              Waypoint Home3: TCP in base x=-850.182 y=0 z=211.32 mm, rx=-2.0297 ry=2.3968 rz=0.0066 rad; joints [-14.374, -75.698, 98.757, -22.649, -284.037, -0.192] deg; TCP offset x=0.411 y=-218.298 z=37.994 mm, rx=1.558 ry=-0.1255 rz=0.1212 rad
              Waypoint Linea4_A: TCP in base x=-486.109 y=25.046 z=110.758 mm, rx=-2.0297 ry=2.3968 rz=0.0065 rad; joints [-35.513, -108.192, 141.382, -32.663, -305.184, -0.389] deg; TCP offset x=0.411 y=-218.298 z=37.994 mm, rx=1.558 ry=-0.1255 rz=0.1212 rad
              Waypoint Linea4_B: TCP in base x=-689.318 y=25.343 z=110.27 mm, rx=-2.0298 ry=2.3969 rz=0.0066 rad; joints [-21.509, -85.16, 121.882, -36.295, -291.196, -0.227] deg
              Waypoint Linea4_C: TCP in base x=-714.721 y=25.086 z=110.565 mm, rx=-2.0298 ry=2.3969 rz=0.0065 rad; joints [-20.482, -82.844, 119.204, -35.936, -290.168, -0.217] deg
              Waypoint Linea4_D: TCP in base x=-918.063 y=25.353 z=110.171 mm, rx=-2.0298 ry=2.3969 rz=0.0065 rad; joints [-14.96, -65.479, 95.824, -29.942, -284.639, -0.166] deg
              Waypoint Linea4_E: TCP in base x=-942.591 y=25.362 z=110.65 mm, rx=-2.0298 ry=2.3969 rz=0.0065 rad; joints [-14.49, -63.451, 92.661, -28.807, -284.167, -0.163] deg
              Waypoint Linea4_F: TCP in base x=-1145.81 y=25.561 z=110.408 mm, rx=-2.0298 ry=2.3969 rz=0.0066 rad; joints [-11.507, -45.055, 61.81, -16.363, -281.155, -0.146] deg
          Folder AB
            'desbaste_inicial'
            bajada_broca := p[0,0,-0.012,0,0,0]
            barrenos_menos1 := 8
            barreno_actual := 0
            Loop While (checkContinuously=false) expression=barreno_actual≤barrenos_menos1
              Folder Perforacion
                MoveL speed 100 mm/s, acceleration 500 mm/s^2 (useActiveTCP=true) feature=Base
                  internos := interpolate_pose(Linea4_A, Linea4_B, barreno_actual/barrenos_menos1)
                  Waypoint Waypoint (Variable): variable=internos
                  'desbaste_inicial'
                  bajada_broca := p[0,0,-0.012,0,0,0]
                  bajada := p[0,0,0.012,0,0,0]
                  MoveDirectionNode (selectedDirection=ZMinus toolParams=0.03, 0.035)
                    Until DISTANCE (allowActions=false deceleration=3 distanceNodeType=STOP) Distance=0.08; motionParameters(blendRadius=0)
                  Popup Message (haltProgram=false message=punto contacto alanzdo inputType=Text)
                  MoveDirectionNode (selectedDirection=ZPlus toolParams=0.003, 0.005)
                    Until DISTANCE (allowActions=false deceleration=3 distanceNodeType=STOP) Distance=0.002; motionParameters(blendRadius=0)
                  Wait Sleep waitTime=0.3
                  Set DigitalOutput pin=config_out[1]; digitalValue=1
                  Wait Sleep waitTime=0.3
                  Loop Counting (count=2) loopVariable(name=Loop_72)
                    bajar := pose_add(get_actual_tcp_pose(), bajada_broca)
                    Waypoint Waypoint (Variable): motionParameters(jointSpeed=1.047198 jointAcceleration=1.396263 cartesianSpeed=0.001 cartesianAcceleration=0.005); variable=bajar
                    subir := pose_sub(get_actual_tcp_pose(), bajada_broca)
                    Waypoint Waypoint (Variable): motionParameters(jointSpeed=1.047198 jointAcceleration=1.396263 cartesianSpeed=0.01 cartesianAcceleration=0.01); variable=subir
                    bajada_broca := pose_sub(bajada_broca, bajada)
                  MoveDirectionNode (selectedDirection=ZPlus toolParams=0.03, 0.035)
                    Until DISTANCE (allowActions=false deceleration=3 distanceNodeType=STOP) Distance=0.06; motionParameters(blendRadius=0)
                  Set DigitalOutput pin=config_out[1]; digitalValue=0
                  barreno_actual := barreno_actual+1
                  Call Quitar_broca
                  Call Poner_broca
          Folder CD
            'desbaste_inicial'
            bajada_broca := p[0,0,-0.012,0,0,0]
            barrenos_menos1 := 8
            barreno_actual := 0
            Loop While (checkContinuously=false) expression=barreno_actual≤barrenos_menos1
              Folder Perforacion
                MoveL speed 100 mm/s, acceleration 500 mm/s^2 (useActiveTCP=true) feature=Base
                  internos := interpolate_pose(Linea4_C, Linea4_D, barreno_actual/barrenos_menos1)
                  Waypoint Waypoint (Variable): variable=internos
                  'desbaste_inicial'
                  bajada_broca := p[0,0,-0.012,0,0,0]
                  bajada := p[0,0,0.012,0,0,0]
                  MoveDirectionNode (selectedDirection=ZMinus toolParams=0.03, 0.035)
                    Until DISTANCE (allowActions=false deceleration=3 distanceNodeType=STOP) Distance=0.08; motionParameters(blendRadius=0)
                  Popup Message (haltProgram=false message=punto contacto alanzdo inputType=Text)
                  MoveDirectionNode (selectedDirection=ZPlus toolParams=0.003, 0.005)
                    Until DISTANCE (allowActions=false deceleration=3 distanceNodeType=STOP) Distance=0.002; motionParameters(blendRadius=0)
                  Wait Sleep waitTime=0.3
                  Set DigitalOutput pin=config_out[1]; digitalValue=1
                  Wait Sleep waitTime=0.3
                  Loop Counting (count=2) loopVariable(name=Loop_77)
                    bajar := pose_add(get_actual_tcp_pose(), bajada_broca)
                    Waypoint Waypoint (Variable): motionParameters(jointSpeed=1.047198 jointAcceleration=1.396263 cartesianSpeed=0.001 cartesianAcceleration=0.005); variable=bajar
                    subir := pose_sub(get_actual_tcp_pose(), bajada_broca)
                    Waypoint Waypoint (Variable): motionParameters(jointSpeed=1.047198 jointAcceleration=1.396263 cartesianSpeed=0.01 cartesianAcceleration=0.01); variable=subir
                    bajada_broca := pose_sub(bajada_broca, bajada)
                  MoveDirectionNode (selectedDirection=ZPlus toolParams=0.03, 0.035)
                    Until DISTANCE (allowActions=false deceleration=3 distanceNodeType=STOP) Distance=0.06; motionParameters(blendRadius=0)
                  Set DigitalOutput pin=config_out[1]; digitalValue=0
                  barreno_actual := barreno_actual+1
                  Call Quitar_broca
                  Call Poner_broca
          Folder EF
            'desbaste_inicial'
            bajada_broca := p[0,0,-0.012,0,0,0]
            barrenos_menos1 := 8
            barreno_actual := 0
            Loop While (checkContinuously=false) expression=barreno_actual≤barrenos_menos1
              Folder Perforacion
                MoveL speed 100 mm/s, acceleration 500 mm/s^2 (useActiveTCP=true) feature=Base
                  internos := interpolate_pose(Linea4_E, Linea4_F, barreno_actual/barrenos_menos1)
                  Waypoint Waypoint (Variable): variable=internos
                  'desbaste_inicial'
                  bajada_broca := p[0,0,-0.012,0,0,0]
                  bajada := p[0,0,0.012,0,0,0]
                  MoveDirectionNode (selectedDirection=ZMinus toolParams=0.03, 0.035)
                    Until DISTANCE (allowActions=false deceleration=3 distanceNodeType=STOP) Distance=0.08; motionParameters(blendRadius=0)
                  Popup Message (haltProgram=false message=punto contacto alanzdo inputType=Text)
                  MoveDirectionNode (selectedDirection=ZPlus toolParams=0.003, 0.005)
                    Until DISTANCE (allowActions=false deceleration=3 distanceNodeType=STOP) Distance=0.002; motionParameters(blendRadius=0)
                  Wait Sleep waitTime=0.3
                  Set DigitalOutput pin=config_out[1]; digitalValue=1
                  Wait Sleep waitTime=0.3
                  Loop Counting (count=2) loopVariable(name=Loop_81)
                    bajar := pose_add(get_actual_tcp_pose(), bajada_broca)
                    Waypoint Waypoint (Variable): motionParameters(jointSpeed=1.047198 jointAcceleration=1.396263 cartesianSpeed=0.001 cartesianAcceleration=0.005); variable=bajar
                    subir := pose_sub(get_actual_tcp_pose(), bajada_broca)
                    Waypoint Waypoint (Variable): motionParameters(jointSpeed=1.047198 jointAcceleration=1.396263 cartesianSpeed=0.01 cartesianAcceleration=0.01); variable=subir
                    bajada_broca := pose_sub(bajada_broca, bajada)
                  MoveDirectionNode (selectedDirection=ZPlus toolParams=0.03, 0.035)
                    Until DISTANCE (allowActions=false deceleration=3 distanceNodeType=STOP) Distance=0.06; motionParameters(blendRadius=0)
                  Set DigitalOutput pin=config_out[1]; digitalValue=0
                  barreno_actual := barreno_actual+1
                  If barreno_actual>barrenos_menos1
                    cambiar_broca := True
                  Call Quitar_broca
                  Call Poner_broca
        Popup Message (haltProgram=false message=Linea4 con media Terminada! inputType=Text)
      Folder Broca_3
        Folder Linea3
          Folder Marcar_puntos
            MoveL speed 100 mm/s, acceleration 500 mm/s^2 (useActiveTCP=true) feature=Base
              Waypoint Home3: TCP in base x=-850.182 y=0 z=211.32 mm, rx=-2.0297 ry=2.3968 rz=0.0066 rad; joints [-14.374, -75.698, 98.757, -22.649, -284.037, -0.192] deg; TCP offset x=0.411 y=-218.298 z=37.994 mm, rx=1.558 ry=-0.1255 rz=0.1212 rad
              Folder var
                barrenos_hechos := 0
                eje7 := 3
                cambiar_broca := False
                iniciando_prog := True
              Call Poner_broca
              Waypoint Linea3_A: TCP in base x=-486.114 y=-381.655 z=110.21 mm, rx=-2.0297 ry=2.3968 rz=0.0065 rad; joints [28.783, -88.014, 124.97, -36.558, -240.905, 0.122] deg; TCP offset x=0.411 y=-218.298 z=37.994 mm, rx=1.558 ry=-0.1255 rz=0.1212 rad
              Waypoint Linea3_B: TCP in base x=-689.31 y=-380.791 z=110.221 mm, rx=-2.0297 ry=2.3969 rz=0.0065 rad; joints [20.056, -74.462, 108.7, -33.857, -249.629, 0.064] deg
              Waypoint Linea3_C: TCP in base x=-714.73 y=-381.227 z=110.547 mm, rx=-2.0298 ry=2.3969 rz=0.0065 rad; joints [19.334, -72.698, 106.253, -33.176, -250.351, 0.061] deg
              Waypoint Linea3_D: TCP in base x=-917.837 y=-380.542 z=110.222 mm, rx=-2.0298 ry=2.3969 rz=0.0065 rad; joints [14.731, -57.949, 83.951, -25.628, -254.939, 0.03] deg
              Waypoint Linea3_E: TCP in base x=-943.23 y=-380.75 z=110.26 mm, rx=-2.0297 ry=2.3969 rz=0.0065 rad; joints [14.315, -55.955, 80.664, -24.335, -255.35, 0.027] deg
              Waypoint Linea3_F: TCP in base x=-1146.085 y=-380.44 z=110.221 mm, rx=-2.0297 ry=2.397 rz=0.0066 rad; joints [11.572, -37.03, 47.136, -9.737, -258.055, 0.004] deg
          Folder AB
            'desbaste_inicial'
            bajada_broca := p[0,0,-0.024,0,0,0]
            barrenos_menos1 := 8
            barreno_actual := 5
            Loop While (checkContinuously=false) expression=barreno_actual≤barrenos_menos1
              Folder Perforacion
                MoveL speed 100 mm/s, acceleration 500 mm/s^2 (useActiveTCP=true) feature=Base
                  internos := interpolate_pose(Linea3_A, Linea3_B, barreno_actual/barrenos_menos1)
                  Waypoint Waypoint (Variable): variable=internos
                  'desbaste_inicial'
                  bajada_broca := p[0,0,-0.024,0,0,0]
                  bajada := p[0,0,0.024,0,0,0]
                  MoveDirectionNode (selectedDirection=ZMinus toolParams=0.03, 0.035)
                    Until DISTANCE (allowActions=false deceleration=3 distanceNodeType=STOP) Distance=0.083; motionParameters(blendRadius=0)
                  Popup Message (haltProgram=false message=punto contacto alanzdo inputType=Text)
                  MoveDirectionNode (selectedDirection=ZPlus toolParams=0.003, 0.005)
                    Until DISTANCE (allowActions=false deceleration=3 distanceNodeType=STOP) Distance=0.002; motionParameters(blendRadius=0)
                  Wait Sleep waitTime=0.3
                  Set DigitalOutput pin=config_out[1]; digitalValue=1
                  Wait Sleep waitTime=0.3
                  Loop Counting (count=1) loopVariable=Loop_86
                    bajar := pose_add(get_actual_tcp_pose(), bajada_broca)
                    Waypoint Waypoint (Variable): motionParameters(jointSpeed=1.047198 jointAcceleration=1.396263 cartesianSpeed=0.001 cartesianAcceleration=0.005); variable=bajar
                    subir := pose_sub(get_actual_tcp_pose(), bajada_broca)
                    Waypoint Waypoint (Variable): motionParameters(jointSpeed=1.047198 jointAcceleration=1.396263 cartesianSpeed=0.01 cartesianAcceleration=0.01); variable=subir
                    bajada_broca := pose_sub(bajada_broca, bajada)
                  MoveDirectionNode (selectedDirection=ZPlus toolParams=0.03, 0.035)
                    Until DISTANCE (allowActions=false deceleration=3 distanceNodeType=STOP) Distance=0.06; motionParameters(blendRadius=0)
                  Set DigitalOutput pin=config_out[1]; digitalValue=0
                  barreno_actual := barreno_actual+1
                  Call Quitar_broca
                  Call Poner_broca
          Folder CD
            'desbaste_inicial'
            bajada_broca := p[0,0,-0.024,0,0,0]
            barrenos_menos1 := 8
            barreno_actual := 0
            Loop While (checkContinuously=false) expression=barreno_actual≤barrenos_menos1
              Folder Perforacion
                MoveL speed 100 mm/s, acceleration 500 mm/s^2 (useActiveTCP=true) feature=Base
                  internos := interpolate_pose(Linea3_C, Linea3_D, barreno_actual/barrenos_menos1)
                  Waypoint Waypoint (Variable): variable=internos
                  'desbaste_inicial'
                  bajada_broca := p[0,0,-0.024,0,0,0]
                  bajada := p[0,0,0.024,0,0,0]
                  MoveDirectionNode (selectedDirection=ZMinus toolParams=0.03, 0.035)
                    Until DISTANCE (allowActions=false deceleration=3 distanceNodeType=STOP) Distance=0.083; motionParameters(blendRadius=0)
                  Popup Message (haltProgram=false message=punto contacto alanzdo inputType=Text)
                  MoveDirectionNode (selectedDirection=ZPlus toolParams=0.003, 0.005)
                    Until DISTANCE (allowActions=false deceleration=3 distanceNodeType=STOP) Distance=0.002; motionParameters(blendRadius=0)
                  Wait Sleep waitTime=0.3
                  Set DigitalOutput pin=config_out[1]; digitalValue=1
                  Wait Sleep waitTime=0.3
                  Loop Counting (count=1) loopVariable(name=Loop_91)
                    bajar := pose_add(get_actual_tcp_pose(), bajada_broca)
                    Waypoint Waypoint (Variable): motionParameters(jointSpeed=1.047198 jointAcceleration=1.396263 cartesianSpeed=0.001 cartesianAcceleration=0.005); variable=bajar
                    subir := pose_sub(get_actual_tcp_pose(), bajada_broca)
                    Waypoint Waypoint (Variable): motionParameters(jointSpeed=1.047198 jointAcceleration=1.396263 cartesianSpeed=0.01 cartesianAcceleration=0.01); variable=subir
                    bajada_broca := pose_sub(bajada_broca, bajada)
                  MoveDirectionNode (selectedDirection=ZPlus toolParams=0.03, 0.035)
                    Until DISTANCE (allowActions=false deceleration=3 distanceNodeType=STOP) Distance=0.06; motionParameters(blendRadius=0)
                  Set DigitalOutput pin=config_out[1]; digitalValue=0
                  barreno_actual := barreno_actual+1
                  Call Quitar_broca
                  Call Poner_broca
          Folder EF
            'desbaste_inicial'
            bajada_broca := p[0,0,-0.024,0,0,0]
            barrenos_menos1 := 8
            barreno_actual := 0
            Loop While (checkContinuously=false) expression=barreno_actual≤barrenos_menos1
              Folder Perforacion
                MoveL speed 100 mm/s, acceleration 500 mm/s^2 (useActiveTCP=true) feature=Base
                  internos := interpolate_pose(Linea3_E, Linea3_F, barreno_actual/barrenos_menos1)
                  Waypoint Waypoint (Variable): variable=internos
                  'desbaste_inicial'
                  bajada_broca := p[0,0,-0.024,0,0,0]
                  bajada := p[0,0,0.024,0,0,0]
                  MoveDirectionNode (selectedDirection=ZMinus toolParams=0.03, 0.035)
                    Until DISTANCE (allowActions=false deceleration=3 distanceNodeType=STOP) Distance=0.083; motionParameters(blendRadius=0)
                  Popup Message (haltProgram=false message=punto contacto alanzdo inputType=Text)
                  MoveDirectionNode (selectedDirection=ZPlus toolParams=0.003, 0.005)
                    Until DISTANCE (allowActions=false deceleration=3 distanceNodeType=STOP) Distance=0.002; motionParameters(blendRadius=0)
                  Wait Sleep waitTime=0.3
                  Set DigitalOutput pin=config_out[1]; digitalValue=1
                  Wait Sleep waitTime=0.3
                  Loop Counting (count=1) loopVariable=Loop_100
                    bajar := pose_add(get_actual_tcp_pose(), bajada_broca)
                    Waypoint Waypoint (Variable): motionParameters(jointSpeed=1.047198 jointAcceleration=1.396263 cartesianSpeed=0.001 cartesianAcceleration=0.005); variable=bajar
                    subir := pose_sub(get_actual_tcp_pose(), bajada_broca)
                    Waypoint Waypoint (Variable): motionParameters(jointSpeed=1.047198 jointAcceleration=1.396263 cartesianSpeed=0.01 cartesianAcceleration=0.01); variable=subir
                    bajada_broca := pose_sub(bajada_broca, bajada)
                  MoveDirectionNode (selectedDirection=ZPlus toolParams=0.03, 0.035)
                    Until DISTANCE (allowActions=false deceleration=3 distanceNodeType=STOP) Distance=0.06; motionParameters(blendRadius=0)
                  Set DigitalOutput pin=config_out[1]; digitalValue=0
                  barreno_actual := barreno_actual+1
                  Call Quitar_broca
                  Call Poner_broca
        Popup Message (haltProgram=false message=Linea3 con full Terminada! inputType=Text)
        Folder Linea4
          Folder Marcar_puntos
            MoveL speed 100 mm/s, acceleration 500 mm/s^2 (useActiveTCP=true) feature=Base
              Waypoint Home3: TCP in base x=-850.182 y=0 z=211.32 mm, rx=-2.0297 ry=2.3968 rz=0.0066 rad; joints [-14.374, -75.698, 98.757, -22.649, -284.037, -0.192] deg; TCP offset x=0.411 y=-218.298 z=37.994 mm, rx=1.558 ry=-0.1255 rz=0.1212 rad
              Waypoint Linea4_A: TCP in base x=-486.109 y=25.046 z=110.758 mm, rx=-2.0297 ry=2.3968 rz=0.0065 rad; joints [-35.513, -108.192, 141.382, -32.663, -305.184, -0.389] deg; TCP offset x=0.411 y=-218.298 z=37.994 mm, rx=1.558 ry=-0.1255 rz=0.1212 rad
              Waypoint Linea4_B: TCP in base x=-689.318 y=25.343 z=110.27 mm, rx=-2.0298 ry=2.3969 rz=0.0066 rad; joints [-21.509, -85.16, 121.882, -36.295, -291.196, -0.227] deg
              Waypoint Linea4_C: TCP in base x=-714.721 y=25.086 z=110.565 mm, rx=-2.0298 ry=2.3969 rz=0.0065 rad; joints [-20.482, -82.844, 119.204, -35.936, -290.168, -0.217] deg
              Waypoint Linea4_D: TCP in base x=-918.063 y=25.353 z=110.171 mm, rx=-2.0298 ry=2.3969 rz=0.0065 rad; joints [-14.96, -65.479, 95.824, -29.942, -284.639, -0.166] deg
              Waypoint Linea4_E: TCP in base x=-942.591 y=25.362 z=110.65 mm, rx=-2.0298 ry=2.3969 rz=0.0065 rad; joints [-14.49, -63.451, 92.661, -28.807, -284.167, -0.163] deg
              Waypoint Linea4_F: TCP in base x=-1145.81 y=25.561 z=110.408 mm, rx=-2.0298 ry=2.3969 rz=0.0066 rad; joints [-11.507, -45.055, 61.81, -16.363, -281.155, -0.146] deg
          Folder AB
            'desbaste_inicial'
            bajada_broca := p[0,0,-0.024,0,0,0]
            barrenos_menos1 := 8
            barreno_actual := 0
            Loop While (checkContinuously=false) expression=barreno_actual≤barrenos_menos1
              Folder Perforacion
                MoveL speed 100 mm/s, acceleration 500 mm/s^2 (useActiveTCP=true) feature=Base
                  internos := interpolate_pose(Linea4_A, Linea4_B, barreno_actual/barrenos_menos1)
                  Waypoint Waypoint (Variable): variable=internos
                  'desbaste_inicial'
                  bajada_broca := p[0,0,-0.024,0,0,0]
                  bajada := p[0,0,0.024,0,0,0]
                  MoveDirectionNode (selectedDirection=ZMinus toolParams=0.03, 0.035)
                    Until DISTANCE (allowActions=false deceleration=3 distanceNodeType=STOP) Distance=0.083; motionParameters(blendRadius=0)
                  Popup Message (haltProgram=false message=punto contacto alanzdo inputType=Text)
                  MoveDirectionNode (selectedDirection=ZPlus toolParams=0.003, 0.005)
                    Until DISTANCE (allowActions=false deceleration=3 distanceNodeType=STOP) Distance=0.002; motionParameters(blendRadius=0)
                  Wait Sleep waitTime=0.3
                  Set DigitalOutput pin=config_out[1]; digitalValue=1
                  Wait Sleep waitTime=0.3
                  Loop Counting (count=1) loopVariable(name=Loop_120)
                    bajar := pose_add(get_actual_tcp_pose(), bajada_broca)
                    Waypoint Waypoint (Variable): motionParameters(jointSpeed=1.047198 jointAcceleration=1.396263 cartesianSpeed=0.001 cartesianAcceleration=0.005); variable=bajar
                    subir := pose_sub(get_actual_tcp_pose(), bajada_broca)
                    Waypoint Waypoint (Variable): motionParameters(jointSpeed=1.047198 jointAcceleration=1.396263 cartesianSpeed=0.01 cartesianAcceleration=0.01); variable=subir
                    bajada_broca := pose_sub(bajada_broca, bajada)
                  MoveDirectionNode (selectedDirection=ZPlus toolParams=0.03, 0.035)
                    Until DISTANCE (allowActions=false deceleration=3 distanceNodeType=STOP) Distance=0.06; motionParameters(blendRadius=0)
                  Set DigitalOutput pin=config_out[1]; digitalValue=0
                  barreno_actual := barreno_actual+1
                  Call Quitar_broca
                  Call Poner_broca
          Folder CD
            'desbaste_inicial'
            bajada_broca := p[0,0,-0.024,0,0,0]
            barrenos_menos1 := 8
            barreno_actual := 0
            Loop While (checkContinuously=false) expression=barreno_actual≤barrenos_menos1
              Folder Perforacion
                MoveL speed 100 mm/s, acceleration 500 mm/s^2 (useActiveTCP=true) feature=Base
                  internos := interpolate_pose(Linea4_C, Linea4_D, barreno_actual/barrenos_menos1)
                  Waypoint Waypoint (Variable): variable=internos
                  'desbaste_inicial'
                  bajada_broca := p[0,0,-0.024,0,0,0]
                  bajada := p[0,0,0.024,0,0,0]
                  MoveDirectionNode (selectedDirection=ZMinus toolParams=0.03, 0.035)
                    Until DISTANCE (allowActions=false deceleration=3 distanceNodeType=STOP) Distance=0.083; motionParameters(blendRadius=0)
                  Popup Message (haltProgram=false message=punto contacto alanzdo inputType=Text)
                  MoveDirectionNode (selectedDirection=ZPlus toolParams=0.003, 0.005)
                    Until DISTANCE (allowActions=false deceleration=3 distanceNodeType=STOP) Distance=0.002; motionParameters(blendRadius=0)
                  Wait Sleep waitTime=0.3
                  Set DigitalOutput pin=config_out[1]; digitalValue=1
                  Wait Sleep waitTime=0.3
                  Loop Counting (count=1) loopVariable=Loop_123
                    bajar := pose_add(get_actual_tcp_pose(), bajada_broca)
                    Waypoint Waypoint (Variable): motionParameters(jointSpeed=1.047198 jointAcceleration=1.396263 cartesianSpeed=0.001 cartesianAcceleration=0.005); variable=bajar
                    subir := pose_sub(get_actual_tcp_pose(), bajada_broca)
                    Waypoint Waypoint (Variable): motionParameters(jointSpeed=1.047198 jointAcceleration=1.396263 cartesianSpeed=0.01 cartesianAcceleration=0.01); variable=subir
                    bajada_broca := pose_sub(bajada_broca, bajada)
                  MoveDirectionNode (selectedDirection=ZPlus toolParams=0.03, 0.035)
                    Until DISTANCE (allowActions=false deceleration=3 distanceNodeType=STOP) Distance=0.06; motionParameters(blendRadius=0)
                  Set DigitalOutput pin=config_out[1]; digitalValue=0
                  barreno_actual := barreno_actual+1
                  Call Quitar_broca
                  Call Poner_broca
          Folder EF
            'desbaste_inicial'
            bajada_broca := p[0,0,-0.024,0,0,0]
            barrenos_menos1 := 8
            barreno_actual := 0
            Loop While (checkContinuously=false) expression=barreno_actual≤barrenos_menos1
              Folder Perforacion
                MoveL speed 100 mm/s, acceleration 500 mm/s^2 (useActiveTCP=true) feature=Base
                  internos := interpolate_pose(Linea4_E, Linea4_F, barreno_actual/barrenos_menos1)
                  Waypoint Waypoint (Variable): variable=internos
                  'desbaste_inicial'
                  bajada_broca := p[0,0,-0.024,0,0,0]
                  bajada := p[0,0,0.024,0,0,0]
                  MoveDirectionNode (selectedDirection=ZMinus toolParams=0.03, 0.035)
                    Until DISTANCE (allowActions=false deceleration=3 distanceNodeType=STOP) Distance=0.083; motionParameters(blendRadius=0)
                  Popup Message (haltProgram=false message=punto contacto alanzdo inputType=Text)
                  MoveDirectionNode (selectedDirection=ZPlus toolParams=0.003, 0.005)
                    Until DISTANCE (allowActions=false deceleration=3 distanceNodeType=STOP) Distance=0.002; motionParameters(blendRadius=0)
                  Wait Sleep waitTime=0.3
                  Set DigitalOutput pin=config_out[1]; digitalValue=1
                  Wait Sleep waitTime=0.3
                  Loop Counting (count=1) loopVariable=Loop_125
                    bajar := pose_add(get_actual_tcp_pose(), bajada_broca)
                    Waypoint Waypoint (Variable): motionParameters(jointSpeed=1.047198 jointAcceleration=1.396263 cartesianSpeed=0.001 cartesianAcceleration=0.005); variable=bajar
                    subir := pose_sub(get_actual_tcp_pose(), bajada_broca)
                    Waypoint Waypoint (Variable): motionParameters(jointSpeed=1.047198 jointAcceleration=1.396263 cartesianSpeed=0.01 cartesianAcceleration=0.01); variable=subir
                    bajada_broca := pose_sub(bajada_broca, bajada)
                  MoveDirectionNode (selectedDirection=ZPlus toolParams=0.03, 0.035)
                    Until DISTANCE (allowActions=false deceleration=3 distanceNodeType=STOP) Distance=0.06; motionParameters(blendRadius=0)
                  Set DigitalOutput pin=config_out[1]; digitalValue=0
                  barreno_actual := barreno_actual+1
                  If barreno_actual>barrenos_menos1
                    cambiar_broca := True
                  Call Quitar_broca
                  Call Poner_broca
        Popup Message (haltProgram=false message=Linea4 con full Terminada! inputType=Text)
    SuppressedNode
      Folder 720
        Folder Broca_1
          Folder Linea5
            Folder Marcar_puntos
              MoveL speed 100 mm/s, acceleration 500 mm/s^2 (useActiveTCP=true) feature=Base
                Waypoint Home3: TCP in base x=-850.182 y=0 z=211.32 mm, rx=-2.0297 ry=2.3968 rz=0.0066 rad; joints [-14.374, -75.698, 98.757, -22.649, -284.037, -0.192] deg; TCP offset x=0.411 y=-218.298 z=37.994 mm, rx=1.558 ry=-0.1255 rz=0.1212 rad
                Waypoint Linea5_A: TCP in base x=-663.778 y=-510.056 z=80.075 mm, rx=3.1116 ry=-0.3921 rz=0.0087 rad; joints [15.224, -65.782, 99.916, -33.468, -339.581, -0.139] deg; TCP offset x=0.411 y=-218.298 z=37.994 mm, rx=1.558 ry=-0.1255 rz=0.1212 rad
                Waypoint Linea5_B: TCP in base x=-1154.197 y=-507.911 z=80.256 mm, rx=-2.6466 ry=1.68 rz=0.0007 rad; joints [13.333, -29.304, 35.323, -5.09, -290.95, -0.372] deg
            Folder AB
              'desbaste_inicial'
              bajada_broca := p[0,0,-0.008,0,0,0]
              barrenos_menos1 := 19
              barreno_actual := 0
              Loop While (checkContinuously=false) expression=barreno_actual≤barrenos_menos1
                Folder Perforacion
                  MoveL speed 100 mm/s, acceleration 500 mm/s^2 (useActiveTCP=true) feature=Base
                    internos := interpolate_pose(Linea5_A, Linea5_B, barreno_actual/barrenos_menos1)
                    Waypoint Waypoint (Variable): variable=internos
                    'desbaste_inicial'
                    bajada_broca := p[0,0,-0.008,0,0,0]
                    bajada := p[0,0,0.008,0,0,0]
                    MoveDirectionNode (selectedDirection=ZMinus toolParams=0.007, 0.005)
                      Until TOOL_CONTACT_DETECTION (allowActions=false retraction=0 decelerationAcceleration=0.001 decelerationAngularAcceleration=34.906585)
                    Popup Message (haltProgram=false message=punto contacto alanzdo inputType=Text)
                    SuppressedNode
                      MoveDirectionNode (selectedDirection=ZPlus toolParams=0.003, 0.005)
                        Until DISTANCE (allowActions=false deceleration=3 distanceNodeType=STOP) Distance=0.002; motionParameters(blendRadius=0)
                    SuppressedNode
                      Wait Sleep waitTime=0.3
                    SuppressedNode
                      Set DigitalOutput pin=config_out[1]; digitalValue=1
                    SuppressedNode
                      Wait Sleep waitTime=0.3
                    SuppressedNode
                      Loop Counting (count=3) loopVariable(name=Loop_55)
                        bajar := pose_add(get_actual_tcp_pose(), bajada_broca)
                        Waypoint Waypoint (Variable): motionParameters(jointSpeed=1.047198 jointAcceleration=1.396263 cartesianSpeed=0.001 cartesianAcceleration=0.005); variable=bajar
                        subir := pose_sub(get_actual_tcp_pose(), bajada_broca)
                        Waypoint Waypoint (Variable): motionParameters(jointSpeed=1.047198 jointAcceleration=1.396263 cartesianSpeed=0.01 cartesianAcceleration=0.01); variable=subir
                        bajada_broca := pose_sub(bajada_broca, bajada)
                    MoveDirectionNode (selectedDirection=ZPlus toolParams=0.03, 0.035)
                      Until DISTANCE (allowActions=false deceleration=3 distanceNodeType=STOP) Distance=0.15; motionParameters(blendRadius=0)
                    Set DigitalOutput pin=config_out[1]; digitalValue=0
                    barreno_actual := barreno_actual+1
                    SuppressedNode
                      Call Quitar_broca
                    SuppressedNode
                      Call Poner_broca
            SuppressedNode
              Folder CD
                'desbaste_inicial'
                bajada_broca := p[0,0,-0.008,0,0,0]
                barrenos_menos1 := 8
                barreno_actual := 0
                Loop While (checkContinuously=false) expression=barreno_actual≤barrenos_menos1
                  Folder Perforacion
                    MoveL speed 100 mm/s, acceleration 500 mm/s^2 (useActiveTCP=true) feature=Base
                      internos := interpolate_pose(Linea3_C, Linea3_D, barreno_actual/barrenos_menos1)
                      Waypoint Waypoint (Variable): variable=internos
                      'desbaste_inicial'
                      bajada_broca := p[0,0,-0.008,0,0,0]
                      bajada := p[0,0,0.008,0,0,0]
                      MoveDirectionNode (selectedDirection=ZMinus toolParams=0.02, 0.015)
                        Until DISTANCE (allowActions=false deceleration=3 distanceNodeType=STOP) Distance=0.055; motionParameters(blendRadius=0)
                      Popup Message (haltProgram=false message=punto contacto alanzdo inputType=Text)
                      MoveDirectionNode (selectedDirection=ZPlus toolParams=0.003, 0.005)
                        Until DISTANCE (allowActions=false deceleration=3 distanceNodeType=STOP) Distance=0.002; motionParameters(blendRadius=0)
                      Wait Sleep waitTime=0.3
                      Set DigitalOutput pin=config_out[1]; digitalValue=1
                      Wait Sleep waitTime=0.3
                      Loop Counting (count=3) loopVariable(name=Loop_57)
                        bajar := pose_add(get_actual_tcp_pose(), bajada_broca)
                        Waypoint Waypoint (Variable): motionParameters(jointSpeed=1.047198 jointAcceleration=1.396263 cartesianSpeed=0.001 cartesianAcceleration=0.005); variable=bajar
                        subir := pose_sub(get_actual_tcp_pose(), bajada_broca)
                        Waypoint Waypoint (Variable): motionParameters(jointSpeed=1.047198 jointAcceleration=1.396263 cartesianSpeed=0.01 cartesianAcceleration=0.01); variable=subir
                        bajada_broca := pose_sub(bajada_broca, bajada)
                      MoveDirectionNode (selectedDirection=ZPlus toolParams=0.03, 0.035)
                        Until DISTANCE (allowActions=false deceleration=3 distanceNodeType=STOP) Distance=0.06; motionParameters(blendRadius=0)
                      Set DigitalOutput pin=config_out[1]; digitalValue=0
                      barreno_actual := barreno_actual+1
                      SuppressedNode
                        Call Quitar_broca
                      SuppressedNode
                        Call Poner_broca
            SuppressedNode
              Folder EF
                'desbaste_inicial'
                bajada_broca := p[0,0,-0.008,0,0,0]
                barrenos_menos1 := 8
                barreno_actual := 0
                Loop While (checkContinuously=false) expression=barreno_actual≤barrenos_menos1
                  Folder Perforacion
                    MoveL speed 100 mm/s, acceleration 500 mm/s^2 (useActiveTCP=true) feature=Base
                      internos := interpolate_pose(Linea3_E, Linea3_F, barreno_actual/barrenos_menos1)
                      Waypoint Waypoint (Variable): variable=internos
                      'desbaste_inicial'
                      bajada_broca := p[0,0,-0.008,0,0,0]
                      bajada := p[0,0,0.008,0,0,0]
                      MoveDirectionNode (selectedDirection=ZMinus toolParams=0.02, 0.015)
                        Until DISTANCE (allowActions=false deceleration=3 distanceNodeType=STOP) Distance=0.055; motionParameters(blendRadius=0)
                      Popup Message (haltProgram=false message=punto contacto alanzdo inputType=Text)
                      MoveDirectionNode (selectedDirection=ZPlus toolParams=0.003, 0.005)
                        Until DISTANCE (allowActions=false deceleration=3 distanceNodeType=STOP) Distance=0.002; motionParameters(blendRadius=0)
                      Wait Sleep waitTime=0.3
                      Set DigitalOutput pin=config_out[1]; digitalValue=1
                      Wait Sleep waitTime=0.3
                      Loop Counting (count=3) loopVariable(name=Loop_59)
                        bajar := pose_add(get_actual_tcp_pose(), bajada_broca)
                        Waypoint Waypoint (Variable): motionParameters(jointSpeed=1.047198 jointAcceleration=1.396263 cartesianSpeed=0.001 cartesianAcceleration=0.005); variable=bajar
                        subir := pose_sub(get_actual_tcp_pose(), bajada_broca)
                        Waypoint Waypoint (Variable): motionParameters(jointSpeed=1.047198 jointAcceleration=1.396263 cartesianSpeed=0.01 cartesianAcceleration=0.01); variable=subir
                        bajada_broca := pose_sub(bajada_broca, bajada)
                      MoveDirectionNode (selectedDirection=ZPlus toolParams=0.03, 0.035)
                        Until DISTANCE (allowActions=false deceleration=3 distanceNodeType=STOP) Distance=0.06; motionParameters(blendRadius=0)
                      Set DigitalOutput pin=config_out[1]; digitalValue=0
                      barreno_actual := barreno_actual+1
                      SuppressedNode
                        Call Quitar_broca
                      SuppressedNode
                        Call Poner_broca
          Popup Message (haltProgram=false message=Linea5 con chica Terminada! inputType=Text)
          Folder Linea6
            Folder Marcar_puntos
              MoveL speed 100 mm/s, acceleration 500 mm/s^2 (useActiveTCP=true) feature=Base
                Waypoint Home3: TCP in base x=-850.182 y=0 z=211.32 mm, rx=-2.0297 ry=2.3968 rz=0.0066 rad; joints [-14.374, -75.698, 98.757, -22.649, -284.037, -0.192] deg; TCP offset x=0.411 y=-218.298 z=37.994 mm, rx=1.558 ry=-0.1255 rz=0.1212 rad
                Waypoint Linea4_A: TCP in base x=-483.35 y=19.133 z=80.413 mm, rx=-2.0297 ry=2.3968 rz=0.0066 rad; joints [-34.857, -105.949, 143.743, -37.281, -304.535, -0.37] deg
                Waypoint Linea4_B: TCP in base x=-685.405 y=19.216 z=80.605 mm, rx=-2.0297 ry=2.3968 rz=0.0066 rad; joints [-21.02, -83.488, 123.782, -39.869, -290.712, -0.217] deg
                Waypoint Linea4_C: TCP in base x=-711.768 y=19.56 z=80.904 mm, rx=-2.0297 ry=2.3968 rz=0.0066 rad; joints [-20.032, -81.151, 120.968, -39.396, -289.723, -0.208] deg
                Waypoint Linea4_D: TCP in base x=-914.58 y=19.801 z=80.703 mm, rx=-2.0297 ry=2.3968 rz=0.0066 rad; joints [-14.612, -64.317, 97.516, -32.795, -284.295, -0.166] deg
                Waypoint Linea4_E: TCP in base x=-939.799 y=20.701 z=80.126 mm, rx=-2.0297 ry=2.3968 rz=0.0066 rad; joints [-14.202, -62.236, 94.311, -31.673, -283.882, -0.163] deg
                Waypoint Linea4_F: TCP in base x=-1143.008 y=20.924 z=80.361 mm, rx=-2.0297 ry=2.3968 rz=0.0066 rad; joints [-11.271, -44.369, 63.742, -18.977, -280.923, -0.147] deg
            Folder AB
              'desbaste_inicial'
              bajada_broca := p[0,0,-0.008,0,0,0]
              barrenos_menos1 := 8
              barreno_actual := 0
              Loop While (checkContinuously=false) expression=barreno_actual≤barrenos_menos1
                Folder Perforacion
                  MoveL speed 100 mm/s, acceleration 500 mm/s^2 (useActiveTCP=true) feature=Base
                    internos := interpolate_pose(Linea4_A, Linea4_B, barreno_actual/barrenos_menos1)
                    Waypoint Waypoint (Variable): variable=internos
                    'desbaste_inicial'
                    bajada_broca := p[0,0,-0.008,0,0,0]
                    bajada := p[0,0,0.008,0,0,0]
                    MoveDirectionNode (selectedDirection=ZMinus toolParams=0.02, 0.015)
                      Until DISTANCE (allowActions=false deceleration=3 distanceNodeType=STOP) Distance=0.055; motionParameters(blendRadius=0)
                    Popup Message (haltProgram=false message=punto contacto alanzdo inputType=Text)
                    MoveDirectionNode (selectedDirection=ZPlus toolParams=0.003, 0.005)
                      Until DISTANCE (allowActions=false deceleration=3 distanceNodeType=STOP) Distance=0.002; motionParameters(blendRadius=0)
                    Wait Sleep waitTime=0.3
                    Set DigitalOutput pin=config_out[1]; digitalValue=1
                    Wait Sleep waitTime=0.3
                    Loop Counting (count=3) loopVariable=Loop_61
                      bajar := pose_add(get_actual_tcp_pose(), bajada_broca)
                      Waypoint Waypoint (Variable): motionParameters(jointSpeed=1.047198 jointAcceleration=1.396263 cartesianSpeed=0.001 cartesianAcceleration=0.005); variable=bajar
                      subir := pose_sub(get_actual_tcp_pose(), bajada_broca)
                      Waypoint Waypoint (Variable): motionParameters(jointSpeed=1.047198 jointAcceleration=1.396263 cartesianSpeed=0.01 cartesianAcceleration=0.01); variable=subir
                      bajada_broca := pose_sub(bajada_broca, bajada)
                    MoveDirectionNode (selectedDirection=ZPlus toolParams=0.03, 0.035)
                      Until DISTANCE (allowActions=false deceleration=3 distanceNodeType=STOP) Distance=0.06; motionParameters(blendRadius=0)
                    Set DigitalOutput pin=config_out[1]; digitalValue=0
                    barreno_actual := barreno_actual+1
                    SuppressedNode
                      Call Quitar_broca
                    SuppressedNode
                      Call Poner_broca
            Folder CD
              'desbaste_inicial'
              bajada_broca := p[0,0,-0.008,0,0,0]
              barrenos_menos1 := 8
              barreno_actual := 0
              Loop While (checkContinuously=false) expression=barreno_actual≤barrenos_menos1
                Folder Perforacion
                  MoveL speed 100 mm/s, acceleration 500 mm/s^2 (useActiveTCP=true) feature=Base
                    internos := interpolate_pose(Linea4_C, Linea4_D, barreno_actual/barrenos_menos1)
                    Waypoint Waypoint (Variable): variable=internos
                    'desbaste_inicial'
                    bajada_broca := p[0,0,-0.008,0,0,0]
                    bajada := p[0,0,0.008,0,0,0]
                    MoveDirectionNode (selectedDirection=ZMinus toolParams=0.02, 0.015)
                      Until DISTANCE (allowActions=false deceleration=3 distanceNodeType=STOP) Distance=0.055; motionParameters(blendRadius=0)
                    Popup Message (haltProgram=false message=punto contacto alanzdo inputType=Text)
                    MoveDirectionNode (selectedDirection=ZPlus toolParams=0.003, 0.005)
                      Until DISTANCE (allowActions=false deceleration=3 distanceNodeType=STOP) Distance=0.002; motionParameters(blendRadius=0)
                    Wait Sleep waitTime=0.3
                    Set DigitalOutput pin=config_out[1]; digitalValue=1
                    Wait Sleep waitTime=0.3
                    Loop Counting (count=3) loopVariable=Loop_63
                      bajar := pose_add(get_actual_tcp_pose(), bajada_broca)
                      Waypoint Waypoint (Variable): motionParameters(jointSpeed=1.047198 jointAcceleration=1.396263 cartesianSpeed=0.001 cartesianAcceleration=0.005); variable=bajar
                      subir := pose_sub(get_actual_tcp_pose(), bajada_broca)
                      Waypoint Waypoint (Variable): motionParameters(jointSpeed=1.047198 jointAcceleration=1.396263 cartesianSpeed=0.01 cartesianAcceleration=0.01); variable=subir
                      bajada_broca := pose_sub(bajada_broca, bajada)
                    MoveDirectionNode (selectedDirection=ZPlus toolParams=0.03, 0.035)
                      Until DISTANCE (allowActions=false deceleration=3 distanceNodeType=STOP) Distance=0.06; motionParameters(blendRadius=0)
                    Set DigitalOutput pin=config_out[1]; digitalValue=0
                    barreno_actual := barreno_actual+1
                    SuppressedNode
                      Call Quitar_broca
                    SuppressedNode
                      Call Poner_broca
            Folder EF
              'desbaste_inicial'
              bajada_broca := p[0,0,-0.008,0,0,0]
              barrenos_menos1 := 8
              barreno_actual := 0
              Loop While (checkContinuously=false) expression=barreno_actual≤barrenos_menos1
                Folder Perforacion
                  MoveL speed 100 mm/s, acceleration 500 mm/s^2 (useActiveTCP=true) feature=Base
                    internos := interpolate_pose(Linea4_E, Linea4_F, barreno_actual/barrenos_menos1)
                    Waypoint Waypoint (Variable): variable=internos
                    'desbaste_inicial'
                    bajada_broca := p[0,0,-0.008,0,0,0]
                    bajada := p[0,0,0.008,0,0,0]
                    MoveDirectionNode (selectedDirection=ZMinus toolParams=0.02, 0.015)
                      Until DISTANCE (allowActions=false deceleration=3 distanceNodeType=STOP) Distance=0.055; motionParameters(blendRadius=0)
                    Popup Message (haltProgram=false message=punto contacto alanzdo inputType=Text)
                    MoveDirectionNode (selectedDirection=ZPlus toolParams=0.003, 0.005)
                      Until DISTANCE (allowActions=false deceleration=3 distanceNodeType=STOP) Distance=0.002; motionParameters(blendRadius=0)
                    Wait Sleep waitTime=0.3
                    Set DigitalOutput pin=config_out[1]; digitalValue=1
                    Wait Sleep waitTime=0.3
                    Loop Counting (count=3) loopVariable=Loop_65
                      bajar := pose_add(get_actual_tcp_pose(), bajada_broca)
                      Waypoint Waypoint (Variable): motionParameters(jointSpeed=1.047198 jointAcceleration=1.396263 cartesianSpeed=0.001 cartesianAcceleration=0.005); variable=bajar
                      subir := pose_sub(get_actual_tcp_pose(), bajada_broca)
                      Waypoint Waypoint (Variable): motionParameters(jointSpeed=1.047198 jointAcceleration=1.396263 cartesianSpeed=0.01 cartesianAcceleration=0.01); variable=subir
                      bajada_broca := pose_sub(bajada_broca, bajada)
                    MoveDirectionNode (selectedDirection=ZPlus toolParams=0.03, 0.035)
                      Until DISTANCE (allowActions=false deceleration=3 distanceNodeType=STOP) Distance=0.06; motionParameters(blendRadius=0)
                    Set DigitalOutput pin=config_out[1]; digitalValue=0
                    barreno_actual := barreno_actual+1
                    If barreno_actual≥barrenos_menos1
                      cambiar_broca := True
                    SuppressedNode
                      Call Quitar_broca
                    SuppressedNode
                      Call Poner_broca
          Popup Message (haltProgram=false message=Linea6 con chica Terminada! inputType=Text)
    Folder 720
      Folder Broca_1
        Folder Linea19
          Folder Marcar_puntos
            MoveL speed 100 mm/s, acceleration 500 mm/s^2 (useActiveTCP=true) feature=Base
              Waypoint Home3: TCP in base x=-850.182 y=0 z=211.32 mm, rx=-2.0297 ry=2.3968 rz=0.0066 rad; joints [-14.374, -75.698, 98.757, -22.649, -284.037, -0.192] deg
              Waypoint Linea19_A: TCP in base x=-476.994 y=-517.247 z=110.482 mm, rx=3.1115 ry=-0.3919 rz=0.0084 rad; joints [20.989, -80.296, 116.237, -35.412, -333.825, -0.009] deg; TCP offset x=0.411 y=-218.298 z=37.994 mm, rx=1.558 ry=-0.1255 rz=0.1212 rad
              Folder bajada_comprobacion
                MoveDirectionNode (selectedDirection=ZMinus toolParams=0.1, 0.15)
                  Until DISTANCE (allowActions=false deceleration=3 distanceNodeType=STOP) Distance=0.071; motionParameters(blendRadius=0)
                MoveDirectionNode (selectedDirection=ZMinus toolParams=0.007, 0.007)
                  Until TOOL_CONTACT_DETECTION (allowActions=false retraction=0 decelerationAcceleration=0.02 decelerationAngularAcceleration=34.906585)
                MoveDirectionNode (selectedDirection=ZPlus toolParams=0.1, 0.15)
                  Until DISTANCE (allowActions=false deceleration=3 distanceNodeType=STOP) Distance=0.08; motionParameters(blendRadius=0)
              Waypoint Linea19_B: TCP in base x=-500.829 y=-517.141 z=110.478 mm, rx=3.1115 ry=-0.3919 rz=0.0084 rad; joints [20.145, -78.637, 114.179, -34.996, -334.668, -0.025] deg
              Folder bajada_comprobacion
                MoveDirectionNode (selectedDirection=ZMinus toolParams=0.1, 0.15)
                  Until DISTANCE (allowActions=false deceleration=3 distanceNodeType=STOP) Distance=0.071; motionParameters(blendRadius=0)
                MoveDirectionNode (selectedDirection=ZMinus toolParams=0.007, 0.007)
                  Until TOOL_CONTACT_DETECTION (allowActions=false retraction=0 decelerationAcceleration=0.02 decelerationAngularAcceleration=34.906585)
                MoveDirectionNode (selectedDirection=ZPlus toolParams=0.1, 0.15)
                  Until DISTANCE (allowActions=false deceleration=3 distanceNodeType=STOP) Distance=0.08; motionParameters(blendRadius=0)
          Folder AB
            'desbaste_inicial'
            bajada_broca := p[0,0,-0.008,0,0,0]
            barrenos_menos1 := 1
            barreno_actual := 0
            Loop While (checkContinuously=false) expression=barreno_actual≤barrenos_menos1
              Folder Perforacion
                MoveL speed 100 mm/s, acceleration 500 mm/s^2 (useActiveTCP=true) feature=Base
                  internos := interpolate_pose(Linea19_A, Linea19_B, barreno_actual/barrenos_menos1)
                  Waypoint Waypoint (Variable): variable=internos
                  'desbaste_inicial'
                  bajada_broca := p[0,0,-0.024,0,0,0]
                  bajada := p[0,0,0.024,0,0,0]
                  MoveDirectionNode (selectedDirection=ZMinus toolParams=0.1, 0.15)
                    Until DISTANCE (allowActions=false deceleration=3 distanceNodeType=STOP) Distance=0.071; motionParameters(blendRadius=0)
                  MoveDirectionNode (selectedDirection=ZMinus toolParams=0.007, 0.007)
                    Until TOOL_CONTACT_DETECTION (allowActions=false retraction=0 decelerationAcceleration=0.02 decelerationAngularAcceleration=34.906585)
                  Popup Message (haltProgram=false message=punto contacto alanzdo inputType=Text)
                  MoveDirectionNode (selectedDirection=ZPlus toolParams=0.015, 0.015)
                    Until DISTANCE (allowActions=false deceleration=3 distanceNodeType=STOP) Distance=0.007; motionParameters(blendRadius=0)
                  Wait Sleep waitTime=0.3
                  Set DigitalOutput pin=config_out[1]; digitalValue=1
                  Wait Sleep waitTime=0.3
                  Loop Counting (count=1) loopVariable=Loop_47
                    bajar := pose_add(get_actual_tcp_pose(), bajada_broca)
                    Waypoint Waypoint (Variable): motionParameters(jointSpeed=1.047198 jointAcceleration=1.396263 cartesianSpeed=0.004 cartesianAcceleration=0.004); variable=bajar
                    subir := pose_sub(get_actual_tcp_pose(), bajada_broca)
                    MoveDirectionNode (selectedDirection=ZPlus toolParams=0.015, 0.015)
                      Until DISTANCE (allowActions=false deceleration=3 distanceNodeType=STOP) Distance=0.002; motionParameters(blendRadius=0)
                    Set DigitalOutput pin=config_out[1]; digitalValue=0
                    Waypoint Waypoint (Variable): motionParameters(jointSpeed=1.047198 jointAcceleration=1.396263 cartesianSpeed=0.015 cartesianAcceleration=0.015); variable=subir
                    bajada_broca := pose_sub(bajada_broca, bajada)
                  MoveDirectionNode (selectedDirection=ZPlus toolParams=0.1, 0.15)
                    Until DISTANCE (allowActions=false deceleration=3 distanceNodeType=STOP) Distance=0.08; motionParameters(blendRadius=0)
                  Set DigitalOutput pin=config_out[1]; digitalValue=0
                  barreno_actual := barreno_actual+1
                  SuppressedNode
                    Call Quitar_broca
                  SuppressedNode
                    Call Poner_broca
        Popup Message (haltProgram=false message=Linea19 con chica Terminada! inputType=Text)
        Folder Linea20
          Folder Marcar_puntos
            MoveL speed 100 mm/s, acceleration 500 mm/s^2 (useActiveTCP=true) feature=Base
              Waypoint Linea20_A: TCP in base x=-530.366 y=-517.559 z=110.808 mm, rx=3.1115 ry=-0.3919 rz=0.0084 rad; joints [19.23, -76.566, 111.483, -34.353, -335.582, -0.045] deg; TCP offset x=0.411 y=-218.298 z=37.994 mm, rx=1.558 ry=-0.1255 rz=0.1212 rad
              Folder bajada_comprobacion
                MoveDirectionNode (selectedDirection=ZMinus toolParams=0.1, 0.15)
                  Until DISTANCE (allowActions=false deceleration=3 distanceNodeType=STOP) Distance=0.071; motionParameters(blendRadius=0)
                MoveDirectionNode (selectedDirection=ZMinus toolParams=0.007, 0.007)
                  Until TOOL_CONTACT_DETECTION (allowActions=false retraction=0 decelerationAcceleration=0.02 decelerationAngularAcceleration=34.906585)
                MoveDirectionNode (selectedDirection=ZPlus toolParams=0.1, 0.15)
                  Until DISTANCE (allowActions=false deceleration=3 distanceNodeType=STOP) Distance=0.08; motionParameters(blendRadius=0)
              Waypoint Linea20_B: TCP in base x=-581.158 y=-517.499 z=110.403 mm, rx=3.1115 ry=-0.3919 rz=0.0084 rad; joints [17.766, -72.963, 106.7, -33.14, -337.045, -0.08] deg
              Folder bajada_comprobacion
                MoveDirectionNode (selectedDirection=ZMinus toolParams=0.1, 0.15)
                  Until DISTANCE (allowActions=false deceleration=3 distanceNodeType=STOP) Distance=0.071; motionParameters(blendRadius=0)
                MoveDirectionNode (selectedDirection=ZMinus toolParams=0.007, 0.007)
                  Until TOOL_CONTACT_DETECTION (allowActions=false retraction=0 decelerationAcceleration=0.02 decelerationAngularAcceleration=34.906585)
                MoveDirectionNode (selectedDirection=ZPlus toolParams=0.1, 0.15)
                  Until DISTANCE (allowActions=false deceleration=3 distanceNodeType=STOP) Distance=0.08; motionParameters(blendRadius=0)
          Folder AB
            'desbaste_inicial'
            bajada_broca := p[0,0,-0.008,0,0,0]
            barrenos_menos1 := 2
            barreno_actual := 0
            Loop While (checkContinuously=false) expression=barreno_actual≤barrenos_menos1
              Folder Perforacion
                MoveL speed 100 mm/s, acceleration 500 mm/s^2 (useActiveTCP=true) feature=Base
                  internos := interpolate_pose(Linea20_A, Linea20_B, barreno_actual/barrenos_menos1)
                  Waypoint Waypoint (Variable): variable=internos
                  'desbaste_inicial'
                  bajada_broca := p[0,0,-0.024,0,0,0]
                  bajada := p[0,0,0.024,0,0,0]
                  MoveDirectionNode (selectedDirection=ZMinus toolParams=0.1, 0.15)
                    Until DISTANCE (allowActions=false deceleration=3 distanceNodeType=STOP) Distance=0.071; motionParameters(blendRadius=0)
                  MoveDirectionNode (selectedDirection=ZMinus toolParams=0.007, 0.007)
                    Until TOOL_CONTACT_DETECTION (allowActions=false retraction=0 decelerationAcceleration=0.02 decelerationAngularAcceleration=34.906585)
                  Popup Message (haltProgram=false message=punto contacto alanzdo inputType=Text)
                  MoveDirectionNode (selectedDirection=ZPlus toolParams=0.015, 0.015)
                    Until DISTANCE (allowActions=false deceleration=3 distanceNodeType=STOP) Distance=0.007; motionParameters(blendRadius=0)
                  Wait Sleep waitTime=0.3
                  Set DigitalOutput pin=config_out[1]; digitalValue=1
                  Wait Sleep waitTime=0.3
                  Loop Counting (count=1) loopVariable=Loop_57
                    bajar := pose_add(get_actual_tcp_pose(), bajada_broca)
                    Waypoint Waypoint (Variable): motionParameters(jointSpeed=1.047198 jointAcceleration=1.396263 cartesianSpeed=0.004 cartesianAcceleration=0.004); variable=bajar
                    subir := pose_sub(get_actual_tcp_pose(), bajada_broca)
                    MoveDirectionNode (selectedDirection=ZPlus toolParams=0.015, 0.015)
                      Until DISTANCE (allowActions=false deceleration=3 distanceNodeType=STOP) Distance=0.002; motionParameters(blendRadius=0)
                    Set DigitalOutput pin=config_out[1]; digitalValue=0
                    Waypoint Waypoint (Variable): motionParameters(jointSpeed=1.047198 jointAcceleration=1.396263 cartesianSpeed=0.015 cartesianAcceleration=0.015); variable=subir
                    bajada_broca := pose_sub(bajada_broca, bajada)
                  MoveDirectionNode (selectedDirection=ZPlus toolParams=0.1, 0.15)
                    Until DISTANCE (allowActions=false deceleration=3 distanceNodeType=STOP) Distance=0.08; motionParameters(blendRadius=0)
                  Set DigitalOutput pin=config_out[1]; digitalValue=0
                  barreno_actual := barreno_actual+1
                  SuppressedNode
                    Call Quitar_broca
                  SuppressedNode
                    Call Poner_broca
        Popup Message (haltProgram=false message=Linea20 con chica Terminada! inputType=Text)
        Folder Linea21
          Folder Marcar_puntos
            MoveL speed 100 mm/s, acceleration 500 mm/s^2 (useActiveTCP=true) feature=Base
              Waypoint Linea21_A: TCP in base x=-665.124 y=-504.211 z=110.6 mm, rx=3.1115 ry=-0.3919 rz=0.0084 rad; joints [14.746, -67.477, 98.83, -30.668, -340.06, -0.171] deg
              Folder bajada_comprobacion
                MoveDirectionNode (selectedDirection=ZMinus toolParams=0.1, 0.15)
                  Until DISTANCE (allowActions=false deceleration=3 distanceNodeType=STOP) Distance=0.071; motionParameters(blendRadius=0)
                MoveDirectionNode (selectedDirection=ZMinus toolParams=0.007, 0.007)
                  Until TOOL_CONTACT_DETECTION (allowActions=false retraction=0 decelerationAcceleration=0.02 decelerationAngularAcceleration=34.906585)
                MoveDirectionNode (selectedDirection=ZPlus toolParams=0.1, 0.15)
                  Until DISTANCE (allowActions=false deceleration=3 distanceNodeType=STOP) Distance=0.08; motionParameters(blendRadius=0)
              SuppressedNode
                Waypoint Linea21_B: TCP in base x=-1156.708 y=-503.073 z=110.552 mm, rx=-2.51 ry=1.8753 rz=0.002 rad; joints [14.221, -30.103, 33.807, -2.778, -281.34, -0.34] deg
              Waypoint Linea21_AB: TCP in base x=-974.251 y=-504.211 z=110.8 mm, rx=3.1115 ry=-0.3919 rz=0.0084 rad; joints [10.309, -41.683, 55.728, -13.152, -344.457, -0.384] deg; TCP offset x=0.411 y=-218.298 z=37.994 mm, rx=1.558 ry=-0.1255 rz=0.1212 rad
              Folder bajada_comprobacion
                MoveDirectionNode (selectedDirection=ZMinus toolParams=0.1, 0.15)
                  Until DISTANCE (allowActions=false deceleration=3 distanceNodeType=STOP) Distance=0.071; motionParameters(blendRadius=0)
                MoveDirectionNode (selectedDirection=ZMinus toolParams=0.007, 0.007)
                  Until TOOL_CONTACT_DETECTION (allowActions=false retraction=0 decelerationAcceleration=0.02 decelerationAngularAcceleration=34.906585)
                MoveDirectionNode (selectedDirection=ZPlus toolParams=0.1, 0.15)
                  Until DISTANCE (allowActions=false deceleration=3 distanceNodeType=STOP) Distance=0.08; motionParameters(blendRadius=0)
          Folder AB
            'desbaste_inicial'
            bajada_broca := p[0,0,-0.008,0,0,0]
            barrenos_menos1 := 12
            barreno_actual := 0
            Loop While (checkContinuously=false) expression=barreno_actual≤barrenos_menos1
              Folder Perforacion
                MoveL speed 100 mm/s, acceleration 500 mm/s^2 (useActiveTCP=true) feature=Base
                  If barreno_actual≟6
                    barreno_actual := barreno_actual+1
                  internos := interpolate_pose(Linea21_A, Linea21_AB, barreno_actual/barrenos_menos1)
                  Waypoint Waypoint (Variable): variable=internos
                  'desbaste_inicial'
                  bajada_broca := p[0,0,-0.024,0,0,0]
                  bajada := p[0,0,0.024,0,0,0]
                  MoveDirectionNode (selectedDirection=ZMinus toolParams=0.1, 0.15)
                    Until DISTANCE (allowActions=false deceleration=3 distanceNodeType=STOP) Distance=0.071; motionParameters(blendRadius=0)
                  MoveDirectionNode (selectedDirection=ZMinus toolParams=0.007, 0.007)
                    Until TOOL_CONTACT_DETECTION (allowActions=false retraction=0 decelerationAcceleration=0.02 decelerationAngularAcceleration=34.906585)
                  Popup Message (haltProgram=false message=punto contacto alanzdo inputType=Text)
                  MoveDirectionNode (selectedDirection=ZPlus toolParams=0.015, 0.015)
                    Until DISTANCE (allowActions=false deceleration=3 distanceNodeType=STOP) Distance=0.007; motionParameters(blendRadius=0)
                  Wait Sleep waitTime=0.3
                  Set DigitalOutput pin=config_out[1]; digitalValue=1
                  Wait Sleep waitTime=0.3
                  Loop Counting (count=1) loopVariable=Loop_76
                    bajar := pose_add(get_actual_tcp_pose(), bajada_broca)
                    Waypoint Waypoint (Variable): motionParameters(jointSpeed=1.047198 jointAcceleration=1.396263 cartesianSpeed=0.004 cartesianAcceleration=0.004); variable=bajar
                    subir := pose_sub(get_actual_tcp_pose(), bajada_broca)
                    MoveDirectionNode (selectedDirection=ZPlus toolParams=0.015, 0.015)
                      Until DISTANCE (allowActions=false deceleration=3 distanceNodeType=STOP) Distance=0.002; motionParameters(blendRadius=0)
                    Set DigitalOutput pin=config_out[1]; digitalValue=0
                    Waypoint Waypoint (Variable): motionParameters(jointSpeed=1.047198 jointAcceleration=1.396263 cartesianSpeed=0.015 cartesianAcceleration=0.015); variable=subir
                    bajada_broca := pose_sub(bajada_broca, bajada)
                  MoveDirectionNode (selectedDirection=ZPlus toolParams=0.1, 0.15)
                    Until DISTANCE (allowActions=false deceleration=3 distanceNodeType=STOP) Distance=0.08; motionParameters(blendRadius=0)
                  Set DigitalOutput pin=config_out[1]; digitalValue=0
                  barreno_actual := barreno_actual+1
                  SuppressedNode
                    Call Quitar_broca
                  SuppressedNode
                    Call Poner_broca
        Popup Message (haltProgram=false message=Linea21 con chica Terminada! inputType=Text)
        Folder Linea21B
          Folder Marcar_puntos
            MoveL speed 100 mm/s, acceleration 500 mm/s^2 (useActiveTCP=true) feature=Base
              SuppressedNode
                Waypoint Linea21_A: TCP in base x=-665.124 y=-504.211 z=110.6 mm, rx=3.1115 ry=-0.3919 rz=0.0084 rad; joints [14.746, -67.477, 98.83, -30.668, -340.06, -0.171] deg; TCP offset x=0.411 y=-218.298 z=37.994 mm, rx=1.558 ry=-0.1255 rz=0.1212 rad
              Waypoint Linea21_BA: TCP in base x=-1025.949 y=-504.193 z=110.366 mm, rx=3.1115 ry=-0.392 rz=0.008 rad; joints [9.807, -35.783, 44.84, -8.147, -344.944, -0.417] deg; TCP offset x=0.411 y=-218.298 z=37.994 mm, rx=1.558 ry=-0.1255 rz=0.1212 rad
              Folder bajada_comprobacion
                MoveDirectionNode (selectedDirection=ZMinus toolParams=0.1, 0.15)
                  Until DISTANCE (allowActions=false deceleration=3 distanceNodeType=STOP) Distance=0.071; motionParameters(blendRadius=0)
                MoveDirectionNode (selectedDirection=ZMinus toolParams=0.007, 0.007)
                  Until TOOL_CONTACT_DETECTION (allowActions=false retraction=0 decelerationAcceleration=0.02 decelerationAngularAcceleration=34.906585)
                MoveDirectionNode (selectedDirection=ZPlus toolParams=0.1, 0.15)
                  Until DISTANCE (allowActions=false deceleration=3 distanceNodeType=STOP) Distance=0.08; motionParameters(blendRadius=0)
              SuppressedNode
                Waypoint Linea21_AB: TCP in base x=-974.251 y=-504.211 z=110.8 mm, rx=3.1115 ry=-0.3919 rz=0.0084 rad; joints [10.309, -41.683, 55.728, -13.152, -344.457, -0.384] deg
              Waypoint Linea21_B: TCP in base x=-1156.708 y=-503.073 z=110.552 mm, rx=-2.51 ry=1.8753 rz=0.002 rad; joints [14.221, -30.103, 33.807, -2.778, -281.34, -0.34] deg; TCP offset x=0.411 y=-218.298 z=37.994 mm, rx=1.558 ry=-0.1255 rz=0.1212 rad
              Folder bajada_comprobacion
                MoveDirectionNode (selectedDirection=ZMinus toolParams=0.1, 0.15)
                  Until DISTANCE (allowActions=false deceleration=3 distanceNodeType=STOP) Distance=0.071; motionParameters(blendRadius=0)
                MoveDirectionNode (selectedDirection=ZMinus toolParams=0.007, 0.007)
                  Until TOOL_CONTACT_DETECTION (allowActions=false retraction=0 decelerationAcceleration=0.02 decelerationAngularAcceleration=34.906585)
                MoveDirectionNode (selectedDirection=ZPlus toolParams=0.1, 0.15)
                  Until DISTANCE (allowActions=false deceleration=3 distanceNodeType=STOP) Distance=0.08; motionParameters(blendRadius=0)
          Folder AB
            'desbaste_inicial'
            bajada_broca := p[0,0,-0.008,0,0,0]
            barrenos_menos1 := 5
            barreno_actual := 0
            Loop While (checkContinuously=false) expression=barreno_actual≤barrenos_menos1
              Folder Perforacion
                MoveL speed 100 mm/s, acceleration 500 mm/s^2 (useActiveTCP=true) feature=Base
                  SuppressedNode
                    If barreno_actual≟6
                      barreno_actual := barreno_actual+1
                  internos := interpolate_pose(Linea21_BA, Linea21_B, barreno_actual/barrenos_menos1)
                  Waypoint Waypoint (Variable): variable=internos
                  'desbaste_inicial'
                  bajada_broca := p[0,0,-0.024,0,0,0]
                  bajada := p[0,0,0.024,0,0,0]
                  MoveDirectionNode (selectedDirection=ZMinus toolParams=0.1, 0.15)
                    Until DISTANCE (allowActions=false deceleration=3 distanceNodeType=STOP) Distance=0.071; motionParameters(blendRadius=0)
                  MoveDirectionNode (selectedDirection=ZMinus toolParams=0.007, 0.007)
                    Until TOOL_CONTACT_DETECTION (allowActions=false retraction=0 decelerationAcceleration=0.02 decelerationAngularAcceleration=34.906585)
                  Popup Message (haltProgram=false message=punto contacto alanzdo inputType=Text)
                  MoveDirectionNode (selectedDirection=ZPlus toolParams=0.015, 0.015)
                    Until DISTANCE (allowActions=false deceleration=3 distanceNodeType=STOP) Distance=0.007; motionParameters(blendRadius=0)
                  Wait Sleep waitTime=0.3
                  Set DigitalOutput pin=config_out[1]; digitalValue=1
                  Wait Sleep waitTime=0.3
                  Loop Counting (count=1) loopVariable(name=Loop_32)
                    bajar := pose_add(get_actual_tcp_pose(), bajada_broca)
                    Waypoint Waypoint (Variable): motionParameters(jointSpeed=1.047198 jointAcceleration=1.396263 cartesianSpeed=0.004 cartesianAcceleration=0.004); variable=bajar
                    subir := pose_sub(get_actual_tcp_pose(), bajada_broca)
                    MoveDirectionNode (selectedDirection=ZPlus toolParams=0.015, 0.015)
                      Until DISTANCE (allowActions=false deceleration=3 distanceNodeType=STOP) Distance=0.002; motionParameters(blendRadius=0)
                    Set DigitalOutput pin=config_out[1]; digitalValue=0
                    Waypoint Waypoint (Variable): motionParameters(jointSpeed=1.047198 jointAcceleration=1.396263 cartesianSpeed=0.015 cartesianAcceleration=0.015); variable=subir
                    bajada_broca := pose_sub(bajada_broca, bajada)
                  MoveDirectionNode (selectedDirection=ZPlus toolParams=0.1, 0.15)
                    Until DISTANCE (allowActions=false deceleration=3 distanceNodeType=STOP) Distance=0.08; motionParameters(blendRadius=0)
                  Set DigitalOutput pin=config_out[1]; digitalValue=0
                  barreno_actual := barreno_actual+1
                  SuppressedNode
                    Call Quitar_broca
                  SuppressedNode
                    Call Poner_broca
        Popup Message (haltProgram=false message=Linea21B con chica Terminada! inputType=Text)
        Folder Linea22
          Folder Marcar_puntos
            MoveL speed 100 mm/s, acceleration 500 mm/s^2 (useActiveTCP=true) feature=Base
              Waypoint Linea22_A: TCP in base x=-637.632 y=-487.983 z=110.98 mm, rx=3.1115 ry=-0.3919 rz=0.0084 rad; joints [14.022, -70.149, 102.677, -31.817, -340.786, -0.198] deg
              Folder bajada_comprobacion
                MoveDirectionNode (selectedDirection=ZMinus toolParams=0.1, 0.15)
                  Until DISTANCE (allowActions=false deceleration=3 distanceNodeType=STOP) Distance=0.071; motionParameters(blendRadius=0)
                MoveDirectionNode (selectedDirection=ZMinus toolParams=0.007, 0.007)
                  Until TOOL_CONTACT_DETECTION (allowActions=false retraction=0 decelerationAcceleration=0.02 decelerationAngularAcceleration=34.906585)
                MoveDirectionNode (selectedDirection=ZPlus toolParams=0.1, 0.15)
                  Until DISTANCE (allowActions=false deceleration=3 distanceNodeType=STOP) Distance=0.08; motionParameters(blendRadius=0)
              Waypoint Linea22_B: TCP in base x=-637.632 y=-461.705 z=110.443 mm, rx=3.1115 ry=-0.3919 rz=0.0084 rad; joints [11.87, -71.111, 104.111, -32.2, -342.939, -0.289] deg
              Folder bajada_comprobacion
                MoveDirectionNode (selectedDirection=ZMinus toolParams=0.1, 0.15)
                  Until DISTANCE (allowActions=false deceleration=3 distanceNodeType=STOP) Distance=0.071; motionParameters(blendRadius=0)
                MoveDirectionNode (selectedDirection=ZMinus toolParams=0.007, 0.007)
                  Until TOOL_CONTACT_DETECTION (allowActions=false retraction=0 decelerationAcceleration=0.02 decelerationAngularAcceleration=34.906585)
                MoveDirectionNode (selectedDirection=ZPlus toolParams=0.1, 0.15)
                  Until DISTANCE (allowActions=false deceleration=3 distanceNodeType=STOP) Distance=0.08; motionParameters(blendRadius=0)
          Folder AB
            'desbaste_inicial'
            bajada_broca := p[0,0,-0.008,0,0,0]
            barrenos_menos1 := 1
            barreno_actual := 0
            Loop While (checkContinuously=false) expression=barreno_actual≤barrenos_menos1
              Folder Perforacion
                MoveL speed 100 mm/s, acceleration 500 mm/s^2 (useActiveTCP=true) feature=Base
                  SuppressedNode
                    If barreno_actual≟6  or barreno_actual≟13
                      barreno_actual := barreno_actual+1
                  internos := interpolate_pose(Linea22_A, Linea22_B, barreno_actual/barrenos_menos1)
                  Waypoint Waypoint (Variable): variable=internos
                  'desbaste_inicial'
                  bajada_broca := p[0,0,-0.024,0,0,0]
                  bajada := p[0,0,0.024,0,0,0]
                  MoveDirectionNode (selectedDirection=ZMinus toolParams=0.1, 0.15)
                    Until DISTANCE (allowActions=false deceleration=3 distanceNodeType=STOP) Distance=0.071; motionParameters(blendRadius=0)
                  MoveDirectionNode (selectedDirection=ZMinus toolParams=0.007, 0.007)
                    Until TOOL_CONTACT_DETECTION (allowActions=false retraction=0 decelerationAcceleration=0.02 decelerationAngularAcceleration=34.906585)
                  Popup Message (haltProgram=false message=punto contacto alanzdo inputType=Text)
                  MoveDirectionNode (selectedDirection=ZPlus toolParams=0.015, 0.015)
                    Until DISTANCE (allowActions=false deceleration=3 distanceNodeType=STOP) Distance=0.007; motionParameters(blendRadius=0)
                  Wait Sleep waitTime=0.3
                  Set DigitalOutput pin=config_out[1]; digitalValue=1
                  Wait Sleep waitTime=0.3
                  Loop Counting (count=1) loopVariable=Loop_84
                    bajar := pose_add(get_actual_tcp_pose(), bajada_broca)
                    Waypoint Waypoint (Variable): motionParameters(jointSpeed=1.047198 jointAcceleration=1.396263 cartesianSpeed=0.004 cartesianAcceleration=0.004); variable=bajar
                    subir := pose_sub(get_actual_tcp_pose(), bajada_broca)
                    MoveDirectionNode (selectedDirection=ZPlus toolParams=0.015, 0.015)
                      Until DISTANCE (allowActions=false deceleration=3 distanceNodeType=STOP) Distance=0.002; motionParameters(blendRadius=0)
                    Set DigitalOutput pin=config_out[1]; digitalValue=0
                    Waypoint Waypoint (Variable): motionParameters(jointSpeed=1.047198 jointAcceleration=1.396263 cartesianSpeed=0.005 cartesianAcceleration=0.01); variable=subir
                    bajada_broca := pose_sub(bajada_broca, bajada)
                  MoveDirectionNode (selectedDirection=ZPlus toolParams=0.1, 0.15)
                    Until DISTANCE (allowActions=false deceleration=3 distanceNodeType=STOP) Distance=0.08; motionParameters(blendRadius=0)
                  Set DigitalOutput pin=config_out[1]; digitalValue=0
                  barreno_actual := barreno_actual+1
                  SuppressedNode
                    Call Quitar_broca
                  SuppressedNode
                    Call Poner_broca
        Popup Message (haltProgram=false message=Linea22 con chica Terminada! inputType=Text)
        Folder Linea23
          Folder Marcar_puntos
            MoveL speed 100 mm/s, acceleration 500 mm/s^2 (useActiveTCP=true) feature=Base
              Waypoint Linea23_A: TCP in base x=-637.535 y=-308.489 z=110.677 mm, rx=3.1115 ry=-0.3919 rz=0.0084 rad; joints [-1.651, -75.077, 109.566, -30.637, -356.453, -3.355] deg
              Folder bajada_comprobacion
                MoveDirectionNode (selectedDirection=ZMinus toolParams=0.1, 0.15)
                  Until DISTANCE (allowActions=false deceleration=3 distanceNodeType=STOP) Distance=0.071; motionParameters(blendRadius=0)
                MoveDirectionNode (selectedDirection=ZMinus toolParams=0.007, 0.007)
                  Until TOOL_CONTACT_DETECTION (allowActions=false retraction=0 decelerationAcceleration=0.02 decelerationAngularAcceleration=34.906585)
                MoveDirectionNode (selectedDirection=ZPlus toolParams=0.1, 0.15)
                  Until DISTANCE (allowActions=false deceleration=3 distanceNodeType=STOP) Distance=0.08; motionParameters(blendRadius=0)
              Waypoint Linea23_B: TCP in base x=-640.734 y=-257.361 z=110.32 mm, rx=-1.9194 ry=2.4833 rz=0.006 rad; joints [10.918, -83.104, 119.505, -35.927, -253.654, -0.007] deg
              Folder bajada_comprobacion
                MoveDirectionNode (selectedDirection=ZMinus toolParams=0.1, 0.15)
                  Until DISTANCE (allowActions=false deceleration=3 distanceNodeType=STOP) Distance=0.071; motionParameters(blendRadius=0)
                MoveDirectionNode (selectedDirection=ZMinus toolParams=0.007, 0.007)
                  Until TOOL_CONTACT_DETECTION (allowActions=false retraction=0 decelerationAcceleration=0.02 decelerationAngularAcceleration=34.906585)
                MoveDirectionNode (selectedDirection=ZPlus toolParams=0.1, 0.15)
                  Until DISTANCE (allowActions=false deceleration=3 distanceNodeType=STOP) Distance=0.08; motionParameters(blendRadius=0)
          Folder AB
            'desbaste_inicial'
            bajada_broca := p[0,0,-0.008,0,0,0]
            barrenos_menos1 := 2
            barreno_actual := 0
            Loop While (checkContinuously=false) expression=barreno_actual≤barrenos_menos1
              Folder Perforacion
                MoveL speed 100 mm/s, acceleration 500 mm/s^2 (useActiveTCP=true) feature=Base
                  SuppressedNode
                    If barreno_actual≟6  or barreno_actual≟13
                      barreno_actual := barreno_actual+1
                  internos := interpolate_pose(Linea23_A, Linea23_B, barreno_actual/barrenos_menos1)
                  Waypoint Waypoint (Variable): variable=internos
                  'desbaste_inicial'
                  bajada_broca := p[0,0,-0.024,0,0,0]
                  bajada := p[0,0,0.024,0,0,0]
                  MoveDirectionNode (selectedDirection=ZMinus toolParams=0.1, 0.15)
                    Until DISTANCE (allowActions=false deceleration=3 distanceNodeType=STOP) Distance=0.071; motionParameters(blendRadius=0)
                  MoveDirectionNode (selectedDirection=ZMinus toolParams=0.007, 0.007)
                    Until TOOL_CONTACT_DETECTION (allowActions=false retraction=0 decelerationAcceleration=0.02 decelerationAngularAcceleration=34.906585)
                  Popup Message (haltProgram=false message=punto contacto alanzdo inputType=Text)
                  MoveDirectionNode (selectedDirection=ZPlus toolParams=0.015, 0.015)
                    Until DISTANCE (allowActions=false deceleration=3 distanceNodeType=STOP) Distance=0.007; motionParameters(blendRadius=0)
                  Wait Sleep waitTime=0.3
                  Set DigitalOutput pin=config_out[1]; digitalValue=1
                  Wait Sleep waitTime=0.3
                  Loop Counting (count=1) loopVariable=Loop_88
                    bajar := pose_add(get_actual_tcp_pose(), bajada_broca)
                    Waypoint Waypoint (Variable): motionParameters(jointSpeed=1.047198 jointAcceleration=1.396263 cartesianSpeed=0.004 cartesianAcceleration=0.004); variable=bajar
                    subir := pose_sub(get_actual_tcp_pose(), bajada_broca)
                    MoveDirectionNode (selectedDirection=ZPlus toolParams=0.015, 0.015)
                      Until DISTANCE (allowActions=false deceleration=3 distanceNodeType=STOP) Distance=0.002; motionParameters(blendRadius=0)
                    Set DigitalOutput pin=config_out[1]; digitalValue=0
                    Waypoint Waypoint (Variable): motionParameters(jointSpeed=1.047198 jointAcceleration=1.396263 cartesianSpeed=0.015 cartesianAcceleration=0.015); variable=subir
                    bajada_broca := pose_sub(bajada_broca, bajada)
                  MoveDirectionNode (selectedDirection=ZPlus toolParams=0.1, 0.15)
                    Until DISTANCE (allowActions=false deceleration=3 distanceNodeType=STOP) Distance=0.08; motionParameters(blendRadius=0)
                  Set DigitalOutput pin=config_out[1]; digitalValue=0
                  barreno_actual := barreno_actual+1
                  SuppressedNode
                    Call Quitar_broca
                  SuppressedNode
                    Call Poner_broca
        Popup Message (haltProgram=false message=Linea23 con chica Terminada! inputType=Text)
        Folder Linea24
          Folder Marcar_puntos
            MoveL speed 100 mm/s, acceleration 500 mm/s^2 (useActiveTCP=true) feature=Base
              Waypoint Linea24_A: TCP in base x=-640.734 y=-233.284 z=110.639 mm, rx=-1.9194 ry=2.4833 rz=0.006 rad; joints [8.334, -84.159, 120.677, -36.046, -256.238, -0.03] deg; TCP offset x=0.411 y=-218.298 z=37.994 mm, rx=1.558 ry=-0.1255 rz=0.1212 rad
              Folder bajada_comprobacion
                MoveDirectionNode (selectedDirection=ZMinus toolParams=0.1, 0.15)
                  Until DISTANCE (allowActions=false deceleration=3 distanceNodeType=STOP) Distance=0.071; motionParameters(blendRadius=0)
                MoveDirectionNode (selectedDirection=ZMinus toolParams=0.007, 0.007)
                  Until TOOL_CONTACT_DETECTION (allowActions=false retraction=0 decelerationAcceleration=0.02 decelerationAngularAcceleration=34.906585)
                MoveDirectionNode (selectedDirection=ZPlus toolParams=0.1, 0.15)
                  Until DISTANCE (allowActions=false deceleration=3 distanceNodeType=STOP) Distance=0.08; motionParameters(blendRadius=0)
              Waypoint Linea24_B: TCP in base x=-640.734 y=-122.85 z=110.749 mm, rx=-1.9194 ry=2.4833 rz=0.006 rad; joints [-4.358, -87.971, 124.826, -36.383, -268.928, -0.138] deg
              Folder bajada_comprobacion
                MoveDirectionNode (selectedDirection=ZMinus toolParams=0.1, 0.15)
                  Until DISTANCE (allowActions=false deceleration=3 distanceNodeType=STOP) Distance=0.071; motionParameters(blendRadius=0)
                MoveDirectionNode (selectedDirection=ZMinus toolParams=0.007, 0.007)
                  Until TOOL_CONTACT_DETECTION (allowActions=false retraction=0 decelerationAcceleration=0.02 decelerationAngularAcceleration=34.906585)
                MoveDirectionNode (selectedDirection=ZPlus toolParams=0.1, 0.15)
                  Until DISTANCE (allowActions=false deceleration=3 distanceNodeType=STOP) Distance=0.08; motionParameters(blendRadius=0)
          Folder AB
            'desbaste_inicial'
            bajada_broca := p[0,0,-0.008,0,0,0]
            barrenos_menos1 := 4
            barreno_actual := 0
            Loop While (checkContinuously=false) expression=barreno_actual≤barrenos_menos1
              Folder Perforacion
                MoveL speed 100 mm/s, acceleration 500 mm/s^2 (useActiveTCP=true) feature=Base
                  If barreno_actual≟2
                    barreno_actual := barreno_actual+1
                  internos := interpolate_pose(Linea24_A, Linea24_B, barreno_actual/barrenos_menos1)
                  Waypoint Waypoint (Variable): variable=internos
                  'desbaste_inicial'
                  bajada_broca := p[0,0,-0.024,0,0,0]
                  bajada := p[0,0,0.024,0,0,0]
                  MoveDirectionNode (selectedDirection=ZMinus toolParams=0.1, 0.15)
                    Until DISTANCE (allowActions=false deceleration=3 distanceNodeType=STOP) Distance=0.071; motionParameters(blendRadius=0)
                  MoveDirectionNode (selectedDirection=ZMinus toolParams=0.007, 0.007)
                    Until TOOL_CONTACT_DETECTION (allowActions=false retraction=0 decelerationAcceleration=0.02 decelerationAngularAcceleration=34.906585)
                  Popup Message (haltProgram=false message=punto contacto alanzdo inputType=Text)
                  MoveDirectionNode (selectedDirection=ZPlus toolParams=0.015, 0.015)
                    Until DISTANCE (allowActions=false deceleration=3 distanceNodeType=STOP) Distance=0.007; motionParameters(blendRadius=0)
                  Wait Sleep waitTime=0.3
                  Set DigitalOutput pin=config_out[1]; digitalValue=1
                  Wait Sleep waitTime=0.3
                  Loop Counting (count=1) loopVariable=Loop_102
                    bajar := pose_add(get_actual_tcp_pose(), bajada_broca)
                    Waypoint Waypoint (Variable): motionParameters(jointSpeed=1.047198 jointAcceleration=1.396263 cartesianSpeed=0.004 cartesianAcceleration=0.004); variable=bajar
                    subir := pose_sub(get_actual_tcp_pose(), bajada_broca)
                    MoveDirectionNode (selectedDirection=ZPlus toolParams=0.015, 0.015)
                      Until DISTANCE (allowActions=false deceleration=3 distanceNodeType=STOP) Distance=0.002; motionParameters(blendRadius=0)
                    Set DigitalOutput pin=config_out[1]; digitalValue=0
                    Waypoint Waypoint (Variable): motionParameters(jointSpeed=1.047198 jointAcceleration=1.396263 cartesianSpeed=0.015 cartesianAcceleration=0.015); variable=subir
                    bajada_broca := pose_sub(bajada_broca, bajada)
                  MoveDirectionNode (selectedDirection=ZPlus toolParams=0.1, 0.15)
                    Until DISTANCE (allowActions=false deceleration=3 distanceNodeType=STOP) Distance=0.08; motionParameters(blendRadius=0)
                  Set DigitalOutput pin=config_out[1]; digitalValue=0
                  barreno_actual := barreno_actual+1
                  SuppressedNode
                    Call Quitar_broca
                  SuppressedNode
                    Call Poner_broca
        Popup Message (haltProgram=false message=Linea24 con chica Terminada! inputType=Text)
        Folder Linea25
          Folder Marcar_puntos
            MoveL speed 100 mm/s, acceleration 500 mm/s^2 (useActiveTCP=true) feature=Base
              Waypoint Linea25_A: TCP in base x=-640.734 y=-99.756 z=110.149 mm, rx=-1.9194 ry=2.4833 rz=0.006 rad; joints [-7.13, -88.49, 125.442, -36.476, -271.701, -0.161] deg; TCP offset x=0.411 y=-218.298 z=37.994 mm, rx=1.558 ry=-0.1255 rz=0.1212 rad
              Folder bajada_comprobacion
                MoveDirectionNode (selectedDirection=ZMinus toolParams=0.1, 0.15)
                  Until DISTANCE (allowActions=false deceleration=3 distanceNodeType=STOP) Distance=0.071; motionParameters(blendRadius=0)
                MoveDirectionNode (selectedDirection=ZMinus toolParams=0.007, 0.007)
                  Until TOOL_CONTACT_DETECTION (allowActions=false retraction=0 decelerationAcceleration=0.02 decelerationAngularAcceleration=34.906585)
                MoveDirectionNode (selectedDirection=ZPlus toolParams=0.1, 0.15)
                  Until DISTANCE (allowActions=false deceleration=3 distanceNodeType=STOP) Distance=0.08; motionParameters(blendRadius=0)
              Waypoint Linea25_B: TCP in base x=-640.734 y=-50.489 z=110.218 mm, rx=-1.9194 ry=2.4833 rz=0.006 rad; joints [-13.081, -89.367, 126.332, -36.479, -277.652, -0.212] deg; TCP offset x=0.411 y=-218.298 z=37.994 mm, rx=1.558 ry=-0.1255 rz=0.1212 rad
              Folder bajada_comprobacion
                MoveDirectionNode (selectedDirection=ZMinus toolParams=0.1, 0.15)
                  Until DISTANCE (allowActions=false deceleration=3 distanceNodeType=STOP) Distance=0.071; motionParameters(blendRadius=0)
                MoveDirectionNode (selectedDirection=ZMinus toolParams=0.007, 0.007)
                  Until TOOL_CONTACT_DETECTION (allowActions=false retraction=0 decelerationAcceleration=0.02 decelerationAngularAcceleration=34.906585)
                MoveDirectionNode (selectedDirection=ZPlus toolParams=0.1, 0.15)
                  Until DISTANCE (allowActions=false deceleration=3 distanceNodeType=STOP) Distance=0.08; motionParameters(blendRadius=0)
          Folder AB
            'desbaste_inicial'
            bajada_broca := p[0,0,-0.008,0,0,0]
            barrenos_menos1 := 2
            barreno_actual := 0
            Loop While (checkContinuously=false) expression=barreno_actual≤barrenos_menos1
              Folder Perforacion
                MoveL speed 100 mm/s, acceleration 500 mm/s^2 (useActiveTCP=true) feature=Base
                  SuppressedNode
                    If barreno_actual≟2
                      barreno_actual := barreno_actual+1
                  internos := interpolate_pose(Linea25_A, Linea25_B, barreno_actual/barrenos_menos1)
                  Waypoint Waypoint (Variable): variable=internos
                  'desbaste_inicial'
                  bajada_broca := p[0,0,-0.024,0,0,0]
                  bajada := p[0,0,0.024,0,0,0]
                  MoveDirectionNode (selectedDirection=ZMinus toolParams=0.1, 0.15)
                    Until DISTANCE (allowActions=false deceleration=3 distanceNodeType=STOP) Distance=0.071; motionParameters(blendRadius=0)
                  MoveDirectionNode (selectedDirection=ZMinus toolParams=0.007, 0.007)
                    Until TOOL_CONTACT_DETECTION (allowActions=false retraction=0 decelerationAcceleration=0.02 decelerationAngularAcceleration=34.906585)
                  Popup Message (haltProgram=false message=punto contacto alanzdo inputType=Text)
                  MoveDirectionNode (selectedDirection=ZPlus toolParams=0.015, 0.015)
                    Until DISTANCE (allowActions=false deceleration=3 distanceNodeType=STOP) Distance=0.007; motionParameters(blendRadius=0)
                  Wait Sleep waitTime=0.3
                  Set DigitalOutput pin=config_out[1]; digitalValue=1
                  Wait Sleep waitTime=0.3
                  Loop Counting (count=1) loopVariable=Loop_135
                    bajar := pose_add(get_actual_tcp_pose(), bajada_broca)
                    Waypoint Waypoint (Variable): motionParameters(jointSpeed=1.047198 jointAcceleration=1.396263 cartesianSpeed=0.004 cartesianAcceleration=0.004); variable=bajar
                    subir := pose_sub(get_actual_tcp_pose(), bajada_broca)
                    MoveDirectionNode (selectedDirection=ZPlus toolParams=0.015, 0.015)
                      Until DISTANCE (allowActions=false deceleration=3 distanceNodeType=STOP) Distance=0.002; motionParameters(blendRadius=0)
                    Set DigitalOutput pin=config_out[1]; digitalValue=0
                    Waypoint Waypoint (Variable): motionParameters(jointSpeed=1.047198 jointAcceleration=1.396263 cartesianSpeed=0.015 cartesianAcceleration=0.015); variable=subir
                    bajada_broca := pose_sub(bajada_broca, bajada)
                  MoveDirectionNode (selectedDirection=ZPlus toolParams=0.1, 0.15)
                    Until DISTANCE (allowActions=false deceleration=3 distanceNodeType=STOP) Distance=0.08; motionParameters(blendRadius=0)
                  Set DigitalOutput pin=config_out[1]; digitalValue=0
                  barreno_actual := barreno_actual+1
                  SuppressedNode
                    Call Quitar_broca
                  SuppressedNode
                    Call Poner_broca
        Popup Message (haltProgram=false message=Linea25 con chica Terminada! inputType=Text)
        Folder Linea26
          Folder Marcar_puntos
            MoveL speed 100 mm/s, acceleration 500 mm/s^2 (useActiveTCP=true) feature=Base
              Waypoint Linea26_A: TCP in base x=-640.548 y=101.33 z=110.865 mm, rx=-1.9194 ry=2.4833 rz=0.006 rad; joints [-30.555, -89.092, 125.972, -36.325, -295.125, -0.376] deg; TCP offset x=0.411 y=-218.298 z=37.994 mm, rx=1.558 ry=-0.1255 rz=0.1212 rad
              Folder bajada_comprobacion
                MoveDirectionNode (selectedDirection=ZMinus toolParams=0.1, 0.15)
                  Until DISTANCE (allowActions=false deceleration=3 distanceNodeType=STOP) Distance=0.071; motionParameters(blendRadius=0)
                MoveDirectionNode (selectedDirection=ZMinus toolParams=0.007, 0.007)
                  Until TOOL_CONTACT_DETECTION (allowActions=false retraction=0 decelerationAcceleration=0.02 decelerationAngularAcceleration=34.906585)
                MoveDirectionNode (selectedDirection=ZPlus toolParams=0.1, 0.15)
                  Until DISTANCE (allowActions=false deceleration=3 distanceNodeType=STOP) Distance=0.08; motionParameters(blendRadius=0)
              Waypoint Linea26_B: TCP in base x=-640.681 y=126.812 z=110.399 mm, rx=-1.9194 ry=2.4833 rz=0.006 rad; joints [-33.193, -88.546, 125.469, -36.353, -297.762, -0.405] deg; TCP offset x=0.411 y=-218.298 z=37.994 mm, rx=1.558 ry=-0.1255 rz=0.1212 rad
              Folder bajada_comprobacion
                MoveDirectionNode (selectedDirection=ZMinus toolParams=0.1, 0.15)
                  Until DISTANCE (allowActions=false deceleration=3 distanceNodeType=STOP) Distance=0.071; motionParameters(blendRadius=0)
                MoveDirectionNode (selectedDirection=ZMinus toolParams=0.007, 0.007)
                  Until TOOL_CONTACT_DETECTION (allowActions=false retraction=0 decelerationAcceleration=0.02 decelerationAngularAcceleration=34.906585)
                MoveDirectionNode (selectedDirection=ZPlus toolParams=0.1, 0.15)
                  Until DISTANCE (allowActions=false deceleration=3 distanceNodeType=STOP) Distance=0.08; motionParameters(blendRadius=0)
          Folder AB
            'desbaste_inicial'
            bajada_broca := p[0,0,-0.008,0,0,0]
            barrenos_menos1 := 1
            barreno_actual := 0
            Loop While (checkContinuously=false) expression=barreno_actual≤barrenos_menos1
              Folder Perforacion
                MoveL speed 100 mm/s, acceleration 500 mm/s^2 (useActiveTCP=true) feature=Base
                  SuppressedNode
                    If barreno_actual≟2
                      barreno_actual := barreno_actual+1
                  internos := interpolate_pose(Linea26_A, Linea26_B, barreno_actual/barrenos_menos1)
                  Waypoint Waypoint (Variable): variable=internos
                  'desbaste_inicial'
                  bajada_broca := p[0,0,-0.024,0,0,0]
                  bajada := p[0,0,0.024,0,0,0]
                  MoveDirectionNode (selectedDirection=ZMinus toolParams=0.1, 0.15)
                    Until DISTANCE (allowActions=false deceleration=3 distanceNodeType=STOP) Distance=0.071; motionParameters(blendRadius=0)
                  MoveDirectionNode (selectedDirection=ZMinus toolParams=0.007, 0.007)
                    Until TOOL_CONTACT_DETECTION (allowActions=false retraction=0 decelerationAcceleration=0.02 decelerationAngularAcceleration=34.906585)
                  Popup Message (haltProgram=false message=punto contacto alanzdo inputType=Text)
                  MoveDirectionNode (selectedDirection=ZPlus toolParams=0.015, 0.015)
                    Until DISTANCE (allowActions=false deceleration=3 distanceNodeType=STOP) Distance=0.007; motionParameters(blendRadius=0)
                  Wait Sleep waitTime=0.3
                  Set DigitalOutput pin=config_out[1]; digitalValue=1
                  Wait Sleep waitTime=0.3
                  Loop Counting (count=1) loopVariable(name=Loop_138)
                    bajar := pose_add(get_actual_tcp_pose(), bajada_broca)
                    Waypoint Waypoint (Variable): motionParameters(jointSpeed=1.047198 jointAcceleration=1.396263 cartesianSpeed=0.004 cartesianAcceleration=0.004); variable=bajar
                    subir := pose_sub(get_actual_tcp_pose(), bajada_broca)
                    MoveDirectionNode (selectedDirection=ZPlus toolParams=0.015, 0.015)
                      Until DISTANCE (allowActions=false deceleration=3 distanceNodeType=STOP) Distance=0.002; motionParameters(blendRadius=0)
                    Set DigitalOutput pin=config_out[1]; digitalValue=0
                    Waypoint Waypoint (Variable): motionParameters(jointSpeed=1.047198 jointAcceleration=1.396263 cartesianSpeed=0.015 cartesianAcceleration=0.015); variable=subir
                    bajada_broca := pose_sub(bajada_broca, bajada)
                  MoveDirectionNode (selectedDirection=ZPlus toolParams=0.1, 0.15)
                    Until DISTANCE (allowActions=false deceleration=3 distanceNodeType=STOP) Distance=0.08; motionParameters(blendRadius=0)
                  Set DigitalOutput pin=config_out[1]; digitalValue=0
                  barreno_actual := barreno_actual+1
                  SuppressedNode
                    Call Quitar_broca
                  SuppressedNode
                    Call Poner_broca
        Popup Message (haltProgram=false message=Linea26 con chica Terminada! inputType=Text)
        Folder Linea27
          Folder Marcar_puntos
            MoveL speed 100 mm/s, acceleration 500 mm/s^2 (useActiveTCP=true) feature=Base
              Waypoint Linea27_A: TCP in base x=-640.02 y=150.733 z=110.213 mm, rx=-1.9194 ry=2.4833 rz=0.006 rad; joints [-35.622, -88.02, 124.944, -36.339, -300.192, -0.432] deg
              Folder bajada_comprobacion
                MoveDirectionNode (selectedDirection=ZMinus toolParams=0.1, 0.15)
                  Until DISTANCE (allowActions=false deceleration=3 distanceNodeType=STOP) Distance=0.071; motionParameters(blendRadius=0)
                MoveDirectionNode (selectedDirection=ZMinus toolParams=0.007, 0.007)
                  Until TOOL_CONTACT_DETECTION (allowActions=false retraction=0 decelerationAcceleration=0.02 decelerationAngularAcceleration=34.906585)
                MoveDirectionNode (selectedDirection=ZPlus toolParams=0.1, 0.15)
                  Until DISTANCE (allowActions=false deceleration=3 distanceNodeType=STOP) Distance=0.08; motionParameters(blendRadius=0)
              Waypoint Linea27_B: TCP in base x=-638.706 y=318.073 z=110.644 mm, rx=0.1163 ry=3.1217 rz=0.0052 rad; joints [-30.379, -75.166, 109.576, -33.746, -215.274, -0.329] deg; TCP offset x=0.411 y=-218.298 z=37.994 mm, rx=1.558 ry=-0.1255 rz=0.1212 rad
              Folder bajada_comprobacion
                MoveDirectionNode (selectedDirection=ZMinus toolParams=0.1, 0.15)
                  Until DISTANCE (allowActions=false deceleration=3 distanceNodeType=STOP) Distance=0.071; motionParameters(blendRadius=0)
                MoveDirectionNode (selectedDirection=ZMinus toolParams=0.007, 0.007)
                  Until TOOL_CONTACT_DETECTION (allowActions=false retraction=0 decelerationAcceleration=0.02 decelerationAngularAcceleration=34.906585)
                MoveDirectionNode (selectedDirection=ZPlus toolParams=0.1, 0.15)
                  Until DISTANCE (allowActions=false deceleration=3 distanceNodeType=STOP) Distance=0.08; motionParameters(blendRadius=0)
          Folder AB
            'desbaste_inicial'
            bajada_broca := p[0,0,-0.008,0,0,0]
            barrenos_menos1 := 6
            barreno_actual := 0
            Loop While (checkContinuously=false) expression=barreno_actual≤barrenos_menos1
              Folder Perforacion
                MoveL speed 100 mm/s, acceleration 500 mm/s^2 (useActiveTCP=true) feature=Base
                  If barreno_actual≟3
                    barreno_actual := barreno_actual+1
                  internos := interpolate_pose(Linea27_A, Linea27_B, barreno_actual/barrenos_menos1)
                  Waypoint Waypoint (Variable): variable=internos
                  'desbaste_inicial'
                  bajada_broca := p[0,0,-0.024,0,0,0]
                  bajada := p[0,0,0.024,0,0,0]
                  MoveDirectionNode (selectedDirection=ZMinus toolParams=0.1, 0.15)
                    Until DISTANCE (allowActions=false deceleration=3 distanceNodeType=STOP) Distance=0.071; motionParameters(blendRadius=0)
                  MoveDirectionNode (selectedDirection=ZMinus toolParams=0.007, 0.007)
                    Until TOOL_CONTACT_DETECTION (allowActions=false retraction=0 decelerationAcceleration=0.02 decelerationAngularAcceleration=34.906585)
                  Popup Message (haltProgram=false message=punto contacto alanzdo inputType=Text)
                  MoveDirectionNode (selectedDirection=ZPlus toolParams=0.015, 0.015)
                    Until DISTANCE (allowActions=false deceleration=3 distanceNodeType=STOP) Distance=0.007; motionParameters(blendRadius=0)
                  Wait Sleep waitTime=0.3
                  Set DigitalOutput pin=config_out[1]; digitalValue=1
                  Wait Sleep waitTime=0.3
                  Loop Counting (count=1) loopVariable(name=Loop_142)
                    bajar := pose_add(get_actual_tcp_pose(), bajada_broca)
                    Waypoint Waypoint (Variable): motionParameters(jointSpeed=1.047198 jointAcceleration=1.396263 cartesianSpeed=0.004 cartesianAcceleration=0.004); variable=bajar
                    subir := pose_sub(get_actual_tcp_pose(), bajada_broca)
                    MoveDirectionNode (selectedDirection=ZPlus toolParams=0.015, 0.015)
                      Until DISTANCE (allowActions=false deceleration=3 distanceNodeType=STOP) Distance=0.002; motionParameters(blendRadius=0)
                    Set DigitalOutput pin=config_out[1]; digitalValue=0
                    Waypoint Waypoint (Variable): motionParameters(jointSpeed=1.047198 jointAcceleration=1.396263 cartesianSpeed=0.015 cartesianAcceleration=0.015); variable=subir
                    bajada_broca := pose_sub(bajada_broca, bajada)
                  MoveDirectionNode (selectedDirection=ZPlus toolParams=0.1, 0.15)
                    Until DISTANCE (allowActions=false deceleration=3 distanceNodeType=STOP) Distance=0.08; motionParameters(blendRadius=0)
                  Set DigitalOutput pin=config_out[1]; digitalValue=0
                  barreno_actual := barreno_actual+1
                  SuppressedNode
                    Call Quitar_broca
                  SuppressedNode
                    Call Poner_broca
        Popup Message (haltProgram=false message=Linea27 con chica Terminada! inputType=Text)
        Folder Linea28
          Folder Marcar_puntos
            MoveL speed 100 mm/s, acceleration 500 mm/s^2 (useActiveTCP=true) feature=Base
